   1:  PR[91,3] = PR[90,3] + 124.000;
   1:L PR[91] R[100]mm/sec CNT100;
   1:  PR[91,1] = PR[90,1] + 30.028;
   1:  PR[91,2] = PR[90,2] + -32.892;
   1:  PR[91,3] = PR[90,3] + 124.033;
   1:L PR[91] R[100]mm/sec CNT100;
   1:  PR[91,1] = PR[90,1] + 35.963;
   1:  PR[91,2] = PR[90,2] + -33.565;
   1:  PR[91,3] = PR[90,3] + 124.037;
   1:L PR[91] R[100]mm/sec CNT100;
   1:  PR[91,1] = PR[90,1] + 39.201;
   1:  PR[91,2] = PR[90,2] + -33.483;
   1:  PR[91,3] = PR[90,3] + 124.069;
   1:L PR[91] R[100]mm/sec CNT100;
   1:  PR[91,1] = PR[90,1] + 41.469;
   1:  PR[91,2] = PR[90,2] + -33.515;
   1:  PR[91,3] = PR[90,3] + 124.087;
   1:L PR[91] R[100]mm/sec CNT100;
   1:  PR[91,1] = PR[90,1] + 46.063;
   1:  PR[91,2] = PR[90,2] + -32.960;
   1:  PR[91,3] = PR[90,3] + 124.100;
   1:L PR[91] R[100]mm/sec CNT100;
   1:  PR[91,1] = PR[90,1] + 51.110;
   1:  PR[91,2] = PR[90,2] + -31.758;
   1:  PR[91,3] = PR[90,3] + 124.125;
   1:L PR[91] R[100]mm/sec CNT100;
   1:  PR[91,1] = PR[90,1] + 55.094;
   1:  PR[91,2] = PR[90,2] + -30.275;
   1:  PR[91,3] = PR[90,3] + 124.154;
   1:L PR[91] R[100]mm/sec CNT100;
   1:  PR[91,1] = PR[90,1] + 56.952;
   1:  PR[91,2] = PR[90,2] + -29.564;
   1:  PR[91,3] = PR[90,3] + 124.177;
   1:L PR[91] R[100]mm/sec CNT100;
   1:  PR[91,1] = PR[90,1] + 60.634;
   1:  PR[91,2] = PR[90,2] + -27.680;
   1:  PR[91,3] = PR[90,3] + 124.188;
   1:L PR[91] R[100]mm/sec CNT100;
   1:  PR[91,1] = PR[90,1] + 63.603;
   1:  PR[91,2] = PR[90,2] + -25.642;
   1:  PR[91,3] = PR[90,3] + 124.211;
   1:L PR[91] R[100]mm/sec CNT100;
   1:  PR[91,1] = PR[90,1] + 65.936;
   1:  PR[91,2] = PR[90,2] + -23.984;
   1:  PR[91,3] = PR[90,3] + 124.231;
   1:L PR[91] R[100]mm/sec CNT100;
   1:  PR[91,1] = PR[90,1] + 68.476;
   1:  PR[91,2] = PR[90,2] + -21.706;
   1:  PR[91,3] = PR[90,3] + 124.247;
   1:L PR[91] R[100]mm/sec CNT100;
   1:  PR[91,1] = PR[90,1] + 70.481;
   1:  PR[91,2] = PR[90,2] + -19.318;
   1:  PR[91,3] = PR[90,3] + 124.265;
   1:L PR[91] R[100]mm/sec CNT100;
   1:  PR[91,1] = PR[90,1] + 72.483;
   1:  PR[91,2] = PR[90,2] + -16.900;
   1:  PR[91,3] = PR[90,3] + 124.282;
   1:L PR[91] R[100]mm/sec CNT100;
   1:  PR[91,1] = PR[90,1] + 74.009;
   1:  PR[91,2] = PR[90,2] + -14.439;
   1:  PR[91,3] = PR[90,3] + 124.300;
   1:L PR[91] R[100]mm/sec CNT100;
   1:  PR[91,1] = PR[90,1] + 75.113;
   1:  PR[91,2] = PR[90,2] + -11.830;
   1:  PR[91,3] = PR[90,3] + 124.316;
   1:L PR[91] R[100]mm/sec CNT100;
   1:  PR[91,1] = PR[90,1] + 76.392;
   1:  PR[91,2] = PR[90,2] + -8.966;
   1:  PR[91,3] = PR[90,3] + 124.331;
   1:L PR[91] R[100]mm/sec CNT100;
   1:  PR[91,1] = PR[90,1] + 77.017;
   1:  PR[91,2] = PR[90,2] + -6.453;
   1:  PR[91,3] = PR[90,3] + 124.349;
   1:L PR[91] R[100]mm/sec CNT100;
   1:  PR[91,1] = PR[90,1] + 77.241;
   1:  PR[91,2] = PR[90,2] + -3.694;
   1:  PR[91,3] = PR[90,3] + 124.363;
   1:L PR[91] R[100]mm/sec CNT100;
   1:  PR[91,1] = PR[90,1] + 77.670;
   1:  PR[91,2] = PR[90,2] + -0.670;
   1:  PR[91,3] = PR[90,3] + 124.378;
   1:L PR[91] R[100]mm/sec CNT100;
   1:  PR[91,1] = PR[90,1] + 77.457;
   1:  PR[91,2] = PR[90,2] + 1.932;
   1:  PR[91,3] = PR[90,3] + 124.395;
   1:L PR[91] R[100]mm/sec CNT100;
   1:  PR[91,1] = PR[90,1] + 77.031;
   1:  PR[91,2] = PR[90,2] + 4.936;
   1:  PR[91,3] = PR[90,3] + 124.409;
   1:L PR[91] R[100]mm/sec CNT100;
   1:  PR[91,1] = PR[90,1] + 76.387;
   1:  PR[91,2] = PR[90,2] + 7.526;
   1:  PR[91,3] = PR[90,3] + 124.426;
   1:L PR[91] R[100]mm/sec CNT100;
   1:  PR[91,1] = PR[90,1] + 75.251;
   1:  PR[91,2] = PR[90,2] + 10.206;
   1:  PR[91,3] = PR[90,3] + 124.441;
   1:L PR[91] R[100]mm/sec CNT100;
   1:  PR[91,1] = PR[90,1] + 74.019;
   1:  PR[91,2] = PR[90,2] + 12.964;
   1:  PR[91,3] = PR[90,3] + 124.457;
   1:L PR[91] R[100]mm/sec CNT100;
   1:  PR[91,1] = PR[90,1] + 72.487;
   1:  PR[91,2] = PR[90,2] + 15.435;
   1:  PR[91,3] = PR[90,3] + 124.473;
   1:L PR[91] R[100]mm/sec CNT100;
   1:  PR[91,1] = PR[90,1] + 70.311;
   1:  PR[91,2] = PR[90,2] + 18.030;
   1:  PR[91,3] = PR[90,3] + 124.489;
   1:L PR[91] R[100]mm/sec CNT100;
   1:  PR[91,1] = PR[90,1] + 68.471;
   1:  PR[91,2] = PR[90,2] + 20.251;
   1:  PR[91,3] = PR[90,3] + 124.508;
   1:L PR[91] R[100]mm/sec CNT100;
   1:  PR[91,1] = PR[90,1] + 65.947;
   1:  PR[91,2] = PR[90,2] + 22.515;
   1:  PR[91,3] = PR[90,3] + 124.524;
   1:L PR[91] R[100]mm/sec CNT100;
   1:  PR[91,1] = PR[90,1] + 62.564;
   1:  PR[91,2] = PR[90,2] + 24.848;
   1:  PR[91,3] = PR[90,3] + 124.543;
   1:L PR[91] R[100]mm/sec CNT100;
   1:  PR[91,1] = PR[90,1] + 60.621;
   1:  PR[91,2] = PR[90,2] + 26.228;
   1:  PR[91,3] = PR[90,3] + 124.565;
   1:L PR[91] R[100]mm/sec CNT100;
   1:  PR[91,1] = PR[90,1] + 56.958;
   1:  PR[91,2] = PR[90,2] + 28.102;
   1:  PR[91,3] = PR[90,3] + 124.578;
   1:L PR[91] R[100]mm/sec CNT100;
   1:  PR[91,1] = PR[90,1] + 51.107;
   1:  PR[91,2] = PR[90,2] + 30.300;
   1:  PR[91,3] = PR[90,3] + 124.601;
   1:L PR[91] R[100]mm/sec CNT100;
   1:  PR[91,1] = PR[90,1] + 46.063;
   1:  PR[91,2] = PR[90,2] + 31.501;
   1:  PR[91,3] = PR[90,3] + 124.635;
   1:L PR[91] R[100]mm/sec CNT100;
   1:  PR[91,1] = PR[90,1] + 41.435;
   1:  PR[91,2] = PR[90,2] + 32.060;
   1:  PR[91,3] = PR[90,3] + 124.664;
   1:L PR[91] R[100]mm/sec CNT100;
   1:  PR[91,1] = PR[90,1] + 38.543;
   1:  PR[91,2] = PR[90,2] + 32.110;
   1:  PR[91,3] = PR[90,3] + 124.690;
   1:L PR[91] R[100]mm/sec CNT100;
   1:  PR[91,1] = PR[90,1] + 35.988;
   1:  PR[91,3] = PR[90,3] + 124.705;
   1:L PR[91] R[100]mm/sec CNT100;
   1:  PR[91,1] = PR[90,1] + 30.052;
   1:  PR[91,2] = PR[90,2] + 31.436;
   1:  PR[91,3] = PR[90,3] + 124.720;
   1:L PR[91] R[100]mm/sec CNT100;
   1:  PR[91,1] = PR[90,1] + 26.924;
   1:  PR[91,2] = PR[90,2] + 30.690;
   1:  PR[91,3] = PR[90,3] + 124.752;
   1:L PR[91] R[100]mm/sec CNT100;
   1:  PR[91,1] = PR[90,1] + 23.579;
   1:  PR[91,2] = PR[90,2] + 29.862;
   1:  PR[91,3] = PR[90,3] + 124.770;
   1:L PR[91] R[100]mm/sec CNT100;
   1:  PR[91,1] = PR[90,1] + 21.241;
   1:  PR[91,2] = PR[90,2] + 29.032;
   1:  PR[91,3] = PR[90,3] + 124.789;
   1:L PR[91] R[100]mm/sec CNT100;
   1:  PR[91,1] = PR[90,1] + 17.734;
   1:  PR[91,2] = PR[90,2] + 27.634;
   1:  PR[91,3] = PR[90,3] + 124.803;
   1:L PR[91] R[100]mm/sec CNT100;
   1:  PR[91,1] = PR[90,1] + 13.334;
   1:  PR[91,2] = PR[90,2] + 25.268;
   1:  PR[91,3] = PR[90,3] + 124.824;
   1:L PR[91] R[100]mm/sec CNT100;
   1:  PR[91,1] = PR[90,1] + 11.692;
   1:  PR[91,2] = PR[90,2] + 24.472;
   1:  PR[91,3] = PR[90,3] + 124.851;
   1:L PR[91] R[100]mm/sec CNT100;
   1:  PR[91,1] = PR[90,1] + 5.360;
   1:  PR[91,2] = PR[90,2] + 20.090;
   1:  PR[91,3] = PR[90,3] + 124.861;
   1:L PR[91] R[100]mm/sec CNT100;
   1:  PR[91,1] = PR[90,1] + 2.591;
   1:  PR[91,2] = PR[90,2] + 17.341;
   1:  PR[91,3] = PR[90,3] + 124.904;
   1:L PR[91] R[100]mm/sec CNT100;
   1:  PR[91,1] = PR[90,1] + 0.096;
   1:  PR[91,2] = PR[90,2] + 15.373;
   1:  PR[91,3] = PR[90,3] + 124.925;
   1:L PR[91] R[100]mm/sec CNT100;
   1:  PR[91,1] = PR[90,1] + -1.259;
   1:  PR[91,2] = PR[90,2] + 13.948;
   1:  PR[91,3] = PR[90,3] + 124.942;
   1:L PR[91] R[100]mm/sec CNT100;
   1:  PR[91,1] = PR[90,1] + -3.418;
   1:  PR[91,2] = PR[90,2] + 11.410;
   1:  PR[91,3] = PR[90,3] + 124.953;
   1:L PR[91] R[100]mm/sec CNT100;
   1:  PR[91,1] = PR[90,1] + -5.567;
   1:  PR[91,2] = PR[90,2] + 8.096;
   1:  PR[91,3] = PR[90,3] + 124.972;
   1:L PR[91] R[100]mm/sec CNT100;
   1:  PR[91,1] = PR[90,1] + -5.693;
   1:  PR[91,2] = PR[90,2] + 7.837;
   1:  PR[91,3] = PR[90,3] + 124.993;
   1:L PR[91] R[100]mm/sec CNT100;
   1:  PR[91] = PR[90];
   1:  PR[91,1] = PR[90,1] + -5.574;
   1:  PR[91,2] = PR[90,2] + 3.809;
   1:  PR[91,3] = PR[90,3] + 126.295;
   1:L PR[91] R[100]mm/sec CNT100;
   1:  PR[91,1] = PR[90,1] + -6.141;
   1:  PR[91,2] = PR[90,2] + -0.559;
   1:  PR[91,3] = PR[90,3] + 125.014;
   1:L PR[91] R[100]mm/sec CNT100;
   1:  PR[91,1] = PR[90,1] + -6.172;
   1:  PR[91,2] = PR[90,2] + -0.756;
   1:  PR[91,3] = PR[90,3] + 125.038;
   1:L PR[91] R[100]mm/sec CNT100;
   1:  PR[91,1] = PR[90,1] + -5.675;
   1:  PR[91,2] = PR[90,2] + -4.661;
   1:  PR[91,3] = PR[90,3] + 125.039;
   1:L PR[91] R[100]mm/sec CNT100;
   1:  PR[91,1] = PR[90,1] + -5.583;
   1:  PR[91,2] = PR[90,2] + -5.243;
   1:  PR[91,3] = PR[90,3] + 125.061;
   1:L PR[91] R[100]mm/sec CNT100;
   1:  PR[91,1] = PR[90,1] + -4.357;
   1:  PR[91,2] = PR[90,2] + -8.470;
   1:  PR[91,3] = PR[90,3] + 125.065;
   1:L PR[91] R[100]mm/sec CNT100;
   1:  PR[91,1] = PR[90,1] + -3.471;
   1:  PR[91,2] = PR[90,2] + -10.288;
   1:  PR[91,3] = PR[90,3] + 125.084;
   1:L PR[91] R[100]mm/sec CNT100;
   1:  PR[91,1] = PR[90,1] + -2.114;
   1:  PR[91,2] = PR[90,2] + -12.382;
   1:  PR[91,3] = PR[90,3] + 125.095;
   1:L PR[91] R[100]mm/sec CNT100;
   1:  PR[91,1] = PR[90,1] + 1.492;
   1:  PR[91,2] = PR[90,2] + -16.619;
   1:  PR[91,3] = PR[90,3] + 125.109;
   1:L PR[91] R[100]mm/sec CNT100;
   1:  PR[91,1] = PR[90,1] + 1.499;
   1:  PR[91,2] = PR[90,2] + -16.626;
   1:  PR[91,3] = PR[90,3] + 125.139;
   1:L PR[91] R[100]mm/sec CNT100;
   1:  PR[91,1] = PR[90,1] + 1.719;
   1:  PR[91,2] = PR[90,2] + -16.800;
   1:  PR[91,3] = PR[90,3] + 125.140;
   1:L PR[91] R[100]mm/sec CNT100;
   1:  PR[91,1] = PR[90,1] + 6.651;
   1:  PR[91,2] = PR[90,2] + -21.698;
   1:  PR[91,3] = PR[90,3] + 125.141;
   1:L PR[91] R[100]mm/sec CNT100;
   1:  PR[91,1] = PR[90,1] + 12.464;
   1:  PR[91,2] = PR[90,2] + -25.715;
   1:  PR[91,3] = PR[90,3] + 125.180;
   1:L PR[91] R[100]mm/sec CNT100;
   1:  PR[91,1] = PR[90,1] + 12.954;
   1:  PR[91,2] = PR[90,2] + -26.093;
   1:  PR[91,3] = PR[90,3] + 125.219;
   1:L PR[91] R[100]mm/sec CNT100;
   1:  PR[91,1] = PR[90,1] + 13.257;
   1:  PR[91,2] = PR[90,2] + -26.269;
   1:  PR[91,3] = PR[90,3] + 125.222;
   1:L PR[91] R[100]mm/sec CNT100;
   1:  PR[91,1] = PR[90,1] + 18.422;
   1:  PR[91,2] = PR[90,2] + -29.047;
   1:  PR[91,3] = PR[90,3] + 125.224;
   1:L PR[91] R[100]mm/sec CNT100;
   1:  PR[91,1] = PR[90,1] + 23.423;
   1:  PR[91,2] = PR[90,2] + -31.043;
   1:  PR[91,3] = PR[90,3] + 125.257;
   1:L PR[91] R[100]mm/sec CNT100;
   1:  PR[91,1] = PR[90,1] + 24.234;
   1:  PR[91,2] = PR[90,2] + -31.331;
   1:  PR[91,3] = PR[90,3] + 125.286;
   1:L PR[91] R[100]mm/sec CNT100;
   1:  PR[91,1] = PR[90,1] + 29.647;
   1:  PR[91,2] = PR[90,2] + -32.658;
   1:  PR[91,3] = PR[90,3] + 125.291;
   1:L PR[91] R[100]mm/sec CNT100;
   1:  PR[91,1] = PR[90,1] + 30.937;
   1:  PR[91,2] = PR[90,2] + -32.945;
   1:  PR[91,3] = PR[90,3] + 125.322;
   1:L PR[91] R[100]mm/sec CNT100;
   1:  PR[91,1] = PR[90,1] + 36.646;
   1:  PR[91,2] = PR[90,2] + -33.595;
   1:  PR[91,3] = PR[90,3] + 125.329;
   1:L PR[91] R[100]mm/sec CNT100;
   1:  PR[91,1] = PR[90,1] + 38.964;
   1:  PR[91,2] = PR[90,2] + -33.537;
   1:  PR[91,3] = PR[90,3] + 125.361;
   1:L PR[91] R[100]mm/sec CNT100;
   1:  PR[91,1] = PR[90,1] + 41.893;
   1:  PR[91,2] = PR[90,2] + -33.577;
   1:  PR[91,3] = PR[90,3] + 125.374;
   1:L PR[91] R[100]mm/sec CNT100;
   1:  PR[91,1] = PR[90,1] + 46.843;
   1:  PR[91,2] = PR[90,2] + -32.976;
   1:  PR[91,3] = PR[90,3] + 125.390;
   1:L PR[91] R[100]mm/sec CNT100;
   1:  PR[91,1] = PR[90,1] + 47.163;
   1:  PR[91,2] = PR[90,2] + -32.917;
   1:  PR[91,3] = PR[90,3] + 125.418;
   1:L PR[91] R[100]mm/sec CNT100;
   1:  PR[91,1] = PR[90,1] + 51.875;
   1:  PR[91,2] = PR[90,2] + -31.789;
   1:  PR[91,3] = PR[90,3] + 125.420;
   1:L PR[91] R[100]mm/sec CNT100;
   1:  PR[91,1] = PR[90,1] + 55.644;
   1:  PR[91,2] = PR[90,2] + -30.386;
   1:  PR[91,3] = PR[90,3] + 125.447;
   1:L PR[91] R[100]mm/sec CNT100;
   1:  PR[91,1] = PR[90,1] + 57.968;
   1:  PR[91,2] = PR[90,2] + -29.496;
   1:  PR[91,3] = PR[90,3] + 125.469;
   1:L PR[91] R[100]mm/sec CNT100;
   1:  PR[91,1] = PR[90,1] + 61.445;
   1:  PR[91,2] = PR[90,2] + -27.718;
   1:  PR[91,3] = PR[90,3] + 125.483;
   1:L PR[91] R[100]mm/sec CNT100;
   1:  PR[91,1] = PR[90,1] + 64.251;
   1:  PR[91,2] = PR[90,2] + -25.791;
   1:  PR[91,3] = PR[90,3] + 125.504;
   1:L PR[91] R[100]mm/sec CNT100;
   1:  PR[91,1] = PR[90,1] + 66.907;
   1:  PR[91,2] = PR[90,2] + -23.903;
   1:  PR[91,3] = PR[90,3] + 125.523;
   1:L PR[91] R[100]mm/sec CNT100;
   1:  PR[91,1] = PR[90,1] + 69.303;
   1:  PR[91,2] = PR[90,2] + -21.754;
   1:  PR[91,3] = PR[90,3] + 125.541;
   1:L PR[91] R[100]mm/sec CNT100;
   1:  PR[91,1] = PR[90,1] + 71.198;
   1:  PR[91,2] = PR[90,2] + -19.499;
   1:  PR[91,3] = PR[90,3] + 125.559;
   1:L PR[91] R[100]mm/sec CNT100;
   1:  PR[91,1] = PR[90,1] + 73.408;
   1:  PR[91,2] = PR[90,2] + -16.830;
   1:  PR[91,3] = PR[90,3] + 125.575;
   1:L PR[91] R[100]mm/sec CNT100;
   1:  PR[91,1] = PR[90,1] + 74.844;
   1:  PR[91,2] = PR[90,2] + -14.512;
   1:  PR[91,3] = PR[90,3] + 125.594;
   1:L PR[91] R[100]mm/sec CNT100;
   1:  PR[91,1] = PR[90,1] + 75.888;
   1:  PR[91,2] = PR[90,2] + -12.046;
   1:  PR[91,3] = PR[90,3] + 125.610;
   1:L PR[91] R[100]mm/sec CNT100;
   1:  PR[91,1] = PR[90,1] + 77.282;
   1:  PR[91,2] = PR[90,2] + -8.925;
   1:  PR[91,3] = PR[90,3] + 125.624;
   1:L PR[91] R[100]mm/sec CNT100;
   1:  PR[91,1] = PR[90,1] + 77.869;
   1:  PR[91,2] = PR[90,2] + -6.562;
   1:  PR[91,3] = PR[90,3] + 125.643;
   1:L PR[91] R[100]mm/sec CNT100;
   1:  PR[91,1] = PR[90,1] + 78.081;
   1:  PR[91,2] = PR[90,2] + -3.954;
   1:  PR[91,3] = PR[90,3] + 125.657;
   1:L PR[91] R[100]mm/sec CNT100;
   1:  PR[91,1] = PR[90,1] + 78.547;
   1:  PR[91,2] = PR[90,2] + -0.670;
   1:  PR[91,3] = PR[90,3] + 125.671;
   1:L PR[91] R[100]mm/sec CNT100;
   1:  PR[91,1] = PR[90,1] + 78.347;
   1:  PR[91,2] = PR[90,2] + 1.780;
   1:  PR[91,3] = PR[90,3] + 125.690;
   1:L PR[91] R[100]mm/sec CNT100;
   1:  PR[91,1] = PR[90,1] + 77.883;
   1:  PR[91,2] = PR[90,2] + 5.046;
   1:  PR[91,3] = PR[90,3] + 125.703;
   1:L PR[91] R[100]mm/sec CNT100;
   1:  PR[91,1] = PR[90,1] + 77.277;
   1:  PR[91,2] = PR[90,2] + 7.485;
   1:  PR[91,3] = PR[90,3] + 125.722;
   1:L PR[91] R[100]mm/sec CNT100;
   1:  PR[91,1] = PR[90,1] + 76.204;
   1:  PR[91,2] = PR[90,2] + 10.015;
   1:  PR[91,3] = PR[90,3] + 125.735;
   1:L PR[91] R[100]mm/sec CNT100;
   1:  PR[91,1] = PR[90,1] + 74.854;
   1:  PR[91,2] = PR[90,2] + 13.036;
   1:  PR[91,3] = PR[90,3] + 125.751;
   1:L PR[91] R[100]mm/sec CNT100;
   1:  PR[91,1] = PR[90,1] + 73.411;
   1:  PR[91,2] = PR[90,2] + 15.365;
   1:  PR[91,3] = PR[90,3] + 125.769;
   1:L PR[91] R[100]mm/sec CNT100;
   1:  PR[91,1] = PR[90,1] + 71.354;
   1:  PR[91,2] = PR[90,2] + 17.818;
   1:  PR[91,3] = PR[90,3] + 125.784;
   1:L PR[91] R[100]mm/sec CNT100;
   1:  PR[91,1] = PR[90,1] + 69.298;
   1:  PR[91,2] = PR[90,2] + 20.300;
   1:  PR[91,3] = PR[90,3] + 125.802;
   1:L PR[91] R[100]mm/sec CNT100;
   1:  PR[91,1] = PR[90,1] + 66.918;
   1:  PR[91,2] = PR[90,2] + 22.435;
   1:  PR[91,3] = PR[90,3] + 125.820;
   1:L PR[91] R[100]mm/sec CNT100;
   1:  PR[91,1] = PR[90,1] + 63.719;
   1:  PR[91,2] = PR[90,2] + 24.641;
   1:  PR[91,3] = PR[90,3] + 125.837;
   1:L PR[91] R[100]mm/sec CNT100;
   1:  PR[91,1] = PR[90,1] + 61.431;
   1:  PR[91,2] = PR[90,2] + 26.266;
   1:  PR[91,3] = PR[90,3] + 125.859;
   1:L PR[91] R[100]mm/sec CNT100;
   1:  PR[91,1] = PR[90,1] + 57.975;
   1:  PR[91,2] = PR[90,2] + 28.034;
   1:  PR[91,3] = PR[90,3] + 125.875;
   1:L PR[91] R[100]mm/sec CNT100;
   1:  PR[91,1] = PR[90,1] + 53.451;
   1:  PR[91,2] = PR[90,2] + 29.725;
   1:  PR[91,3] = PR[90,3] + 125.896;
   1:L PR[91] R[100]mm/sec CNT100;
   1:  PR[91,1] = PR[90,1] + 51.866;
   1:  PR[91,2] = PR[90,2] + 30.332;
   1:  PR[91,3] = PR[90,3] + 125.923;
   1:L PR[91] R[100]mm/sec CNT100;
   1:  PR[91,1] = PR[90,1] + 47.163;
   1:  PR[91,2] = PR[90,2] + 31.458;
   1:  PR[91,3] = PR[90,3] + 125.932;
   1:L PR[91] R[100]mm/sec CNT100;
   1:  PR[91,1] = PR[90,1] + 46.843;
   1:  PR[91,2] = PR[90,2] + 31.517;
   1:  PR[91,3] = PR[90,3] + 125.959;
   1:L PR[91] R[100]mm/sec CNT100;
   1:  PR[91,1] = PR[90,1] + 41.861;
   1:  PR[91,2] = PR[90,2] + 32.122;
   1:  PR[91,3] = PR[90,3] + 125.961;
   1:L PR[91] R[100]mm/sec CNT100;
   1:  PR[91,1] = PR[90,1] + 40.847;
   1:  PR[91,2] = PR[90,2] + 32.140;
   1:  PR[91,3] = PR[90,3] + 125.989;
   1:L PR[91] R[100]mm/sec CNT100;
   1:  PR[91,1] = PR[90,1] + 36.672;
   1:  PR[91,3] = PR[90,3] + 125.994;
   1:L PR[91] R[100]mm/sec CNT100;
   1:  PR[91,1] = PR[90,1] + 30.961;
   1:  PR[91,2] = PR[90,2] + 31.489;
   1:  PR[91,3] = PR[90,3] + 126.017;
   1:L PR[91] R[100]mm/sec CNT100;
   1:  PR[91,1] = PR[90,1] + 24.238;
   1:  PR[91,2] = PR[90,2] + 29.873;
   1:  PR[91,3] = PR[90,3] + 126.049;
   1:L PR[91] R[100]mm/sec CNT100;
   1:  PR[91,1] = PR[90,1] + 23.437;
   1:  PR[91,2] = PR[90,2] + 29.589;
   1:  PR[91,3] = PR[90,3] + 126.087;
   1:L PR[91] R[100]mm/sec CNT100;
   1:  PR[91,1] = PR[90,1] + 18.430;
   1:  PR[91,2] = PR[90,2] + 27.592;
   1:  PR[91,3] = PR[90,3] + 126.092;
   1:L PR[91] R[100]mm/sec CNT100;
   1:  PR[91,1] = PR[90,1] + 13.273;
   1:  PR[91,2] = PR[90,2] + 24.819;
   1:  PR[91,3] = PR[90,3] + 126.122;
   1:L PR[91] R[100]mm/sec CNT100;
   1:  PR[91,1] = PR[90,1] + 12.963;
   1:  PR[91,2] = PR[90,2] + 24.639;
   1:  PR[91,3] = PR[90,3] + 126.154;
   1:L PR[91] R[100]mm/sec CNT100;
   1:  PR[91,1] = PR[90,1] + 12.464;
   1:  PR[91,2] = PR[90,2] + 24.255;
   1:  PR[91,3] = PR[90,3] + 126.156;
   1:L PR[91] R[100]mm/sec CNT100;
   1:  PR[91,1] = PR[90,1] + 6.655;
   1:  PR[91,2] = PR[90,2] + 20.242;
   1:  PR[91,3] = PR[90,3] + 126.160;
   1:L PR[91] R[100]mm/sec CNT100;
   1:  PR[91,1] = PR[90,1] + 1.719;
   1:  PR[91,2] = PR[90,2] + 15.341;
   1:  PR[91,3] = PR[90,3] + 126.199;
   1:L PR[91] R[100]mm/sec CNT100;
   1:  PR[91,1] = PR[90,1] + 1.499;
   1:  PR[91,2] = PR[90,2] + 15.168;
   1:  PR[91,3] = PR[90,3] + 126.238;
   1:L PR[91] R[100]mm/sec CNT100;
   1:  PR[91,1] = PR[90,1] + 1.492;
   1:  PR[91,2] = PR[90,2] + 15.160;
   1:  PR[91,3] = PR[90,3] + 126.239;
   1:L PR[91] R[100]mm/sec CNT100;
   1:  PR[91,1] = PR[90,1] + -2.114;
   1:  PR[91,2] = PR[90,2] + 10.923;
   1:L PR[91] R[100]mm/sec CNT100;
   1:  PR[91,1] = PR[90,1] + -3.471;
   1:  PR[91,2] = PR[90,2] + 8.829;
   1:  PR[91,3] = PR[90,3] + 126.270;
   1:L PR[91] R[100]mm/sec CNT100;
   1:  PR[91,1] = PR[90,1] + -4.357;
   1:  PR[91,2] = PR[90,2] + 7.011;
   1:  PR[91,3] = PR[90,3] + 126.284;
   1:L PR[91] R[100]mm/sec CNT100;
   1:  PR[91] = PR[90];
   1:  PR[91,1] = PR[90,1] + -3.791;
   1:  PR[91,2] = PR[90,2] + 4.159;
   1:  PR[91,3] = PR[90,3] + 127.595;
   1:L PR[91] R[100]mm/sec CNT100;
   1:  PR[91,1] = PR[90,1] + -4.159;
   1:  PR[91,2] = PR[90,2] + 1.325;
   1:  PR[91,3] = PR[90,3] + 126.307;
   1:L PR[91] R[100]mm/sec CNT100;
   1:  PR[91,1] = PR[90,1] + -4.481;
   1:  PR[91,2] = PR[90,2] + -0.756;
   1:  PR[91,3] = PR[90,3] + 126.323;
   1:L PR[91] R[100]mm/sec CNT100;
   1:  PR[91,1] = PR[90,1] + -4.146;
   1:  PR[91,2] = PR[90,2] + -3.392;
   1:  PR[91,3] = PR[90,3] + 126.335;
   1:L PR[91] R[100]mm/sec CNT100;
   1:  PR[91,1] = PR[90,1] + -3.801;
   1:  PR[91,2] = PR[90,2] + -5.593;
   1:  PR[91,3] = PR[90,3] + 126.349;
   1:L PR[91] R[100]mm/sec CNT100;
   1:  PR[91,1] = PR[90,1] + -3.021;
   1:  PR[91,2] = PR[90,2] + -7.644;
   1:  PR[91,3] = PR[90,3] + 126.362;
   1:L PR[91] R[100]mm/sec CNT100;
   1:  PR[91,1] = PR[90,1] + -1.375;
   1:  PR[91,2] = PR[90,2] + -11.021;
   1:  PR[91,3] = PR[90,3] + 126.374;
   1:L PR[91] R[100]mm/sec CNT100;
   1:  PR[91,1] = PR[90,1] + -0.809;
   1:  PR[91,2] = PR[90,2] + -11.894;
   1:  PR[91,3] = PR[90,3] + 126.395;
   1:L PR[91] R[100]mm/sec CNT100;
   1:  PR[91,1] = PR[90,1] + 1.116;
   1:  PR[91,2] = PR[90,2] + -14.156;
   1:  PR[91,3] = PR[90,3] + 126.401;
   1:L PR[91] R[100]mm/sec CNT100;
   1:  PR[91,1] = PR[90,1] + 2.964;
   1:  PR[91,2] = PR[90,2] + -16.913;
   1:  PR[91,3] = PR[90,3] + 126.417;
   1:L PR[91] R[100]mm/sec CNT100;
   1:  PR[91,1] = PR[90,1] + 7.943;
   1:  PR[91,2] = PR[90,2] + -21.848;
   1:  PR[91,3] = PR[90,3] + 126.436;
   1:L PR[91] R[100]mm/sec CNT100;
   1:  PR[91,1] = PR[90,1] + 11.325;
   1:  PR[91,2] = PR[90,2] + -24.184;
   1:  PR[91,3] = PR[90,3] + 126.475;
   1:L PR[91] R[100]mm/sec CNT100;
   1:  PR[91,1] = PR[90,1] + 13.694;
   1:  PR[91,2] = PR[90,2] + -26.010;
   1:  PR[91,3] = PR[90,3] + 126.498;
   1:L PR[91] R[100]mm/sec CNT100;
   1:  PR[91,1] = PR[90,1] + 15.507;
   1:  PR[91,2] = PR[90,2] + -27.063;
   1:  PR[91,3] = PR[90,3] + 126.514;
   1:L PR[91] R[100]mm/sec CNT100;
   1:  PR[91,1] = PR[90,1] + 19.120;
   1:  PR[91,2] = PR[90,2] + -29.006;
   1:  PR[91,3] = PR[90,3] + 126.526;
   1:L PR[91] R[100]mm/sec CNT100;
   1:  PR[91,1] = PR[90,1] + 24.945;
   1:  PR[91,2] = PR[90,2] + -31.339;
   1:  PR[91,3] = PR[90,3] + 126.549;
   1:L PR[91] R[100]mm/sec CNT100;
   1:  PR[91,1] = PR[90,1] + 25.097;
   1:  PR[91,2] = PR[90,2] + -31.390;
   1:  PR[91,3] = PR[90,3] + 126.584;
   1:L PR[91] R[100]mm/sec CNT100;
   1:  PR[91,1] = PR[90,1] + 29.956;
   1:  PR[91,2] = PR[90,2] + -32.577;
   1:  PR[91,3] = PR[90,3] + 126.585;
   1:L PR[91] R[100]mm/sec CNT100;
   1:  PR[91,1] = PR[90,1] + 31.846;
   1:  PR[91,2] = PR[90,2] + -32.998;
   1:  PR[91,3] = PR[90,3] + 126.612;
   1:L PR[91] R[100]mm/sec CNT100;
   1:  PR[91,1] = PR[90,1] + 37.329;
   1:  PR[91,2] = PR[90,2] + -33.626;
   1:  PR[91,3] = PR[90,3] + 126.623;
   1:L PR[91] R[100]mm/sec CNT100;
   1:  PR[91,1] = PR[90,1] + 38.727;
   1:  PR[91,2] = PR[90,2] + -33.590;
   1:  PR[91,3] = PR[90,3] + 126.654;
   1:L PR[91] R[100]mm/sec CNT100;
   1:  PR[91,1] = PR[90,1] + 41.492;
   1:  PR[91,2] = PR[90,2] + -33.628;
   1:  PR[91,3] = PR[90,3] + 126.662;
   1:L PR[91] R[100]mm/sec CNT100;
   1:  PR[91,1] = PR[90,1] + 42.530;
   1:  PR[91,2] = PR[90,2] + -33.612;
   1:  PR[91,3] = PR[90,3] + 126.677;
   1:L PR[91] R[100]mm/sec CNT100;
   1:  PR[91,1] = PR[90,1] + 47.573;
   1:  PR[91,2] = PR[90,2] + -32.998;
   1:  PR[91,3] = PR[90,3] + 126.683;
   1:L PR[91] R[100]mm/sec CNT100;
   1:  PR[91,1] = PR[90,1] + 48.201;
   1:  PR[91,2] = PR[90,2] + -32.882;
   1:  PR[91,3] = PR[90,3] + 126.711;
   1:L PR[91] R[100]mm/sec CNT100;
   1:  PR[91,1] = PR[90,1] + 52.642;
   1:  PR[91,2] = PR[90,2] + -31.819;
   1:  PR[91,3] = PR[90,3] + 126.715;
   1:L PR[91] R[100]mm/sec CNT100;
   1:  PR[91,1] = PR[90,1] + 56.194;
   1:  PR[91,2] = PR[90,2] + -30.497;
   1:  PR[91,3] = PR[90,3] + 126.740;
   1:L PR[91] R[100]mm/sec CNT100;
   1:  PR[91,1] = PR[90,1] + 58.984;
   1:  PR[91,2] = PR[90,2] + -29.429;
   1:  PR[91,3] = PR[90,3] + 126.761;
   1:L PR[91] R[100]mm/sec CNT100;
   1:  PR[91,1] = PR[90,1] + 62.255;
   1:  PR[91,2] = PR[90,2] + -27.755;
   1:  PR[91,3] = PR[90,3] + 126.778;
   1:L PR[91] R[100]mm/sec CNT100;
   1:  PR[91,1] = PR[90,1] + 64.899;
   1:  PR[91,2] = PR[90,2] + -25.940;
   1:  PR[91,3] = PR[90,3] + 126.798;
   1:L PR[91] R[100]mm/sec CNT100;
   1:  PR[91,1] = PR[90,1] + 67.879;
   1:  PR[91,2] = PR[90,2] + -23.823;
   1:  PR[91,3] = PR[90,3] + 126.816;
   1:L PR[91] R[100]mm/sec CNT100;
   1:  PR[91,1] = PR[90,1] + 70.131;
   1:  PR[91,2] = PR[90,2] + -21.803;
   1:  PR[91,3] = PR[90,3] + 126.836;
   1:L PR[91] R[100]mm/sec CNT100;
   1:  PR[91,1] = PR[90,1] + 71.915;
   1:  PR[91,2] = PR[90,2] + -19.678;
   1:  PR[91,3] = PR[90,3] + 126.853;
   1:L PR[91] R[100]mm/sec CNT100;
   1:  PR[91,1] = PR[90,1] + 74.332;
   1:  PR[91,2] = PR[90,2] + -16.759;
   1:  PR[91,3] = PR[90,3] + 126.869;
   1:L PR[91] R[100]mm/sec CNT100;
   1:  PR[91,1] = PR[90,1] + 75.680;
   1:  PR[91,2] = PR[90,2] + -14.584;
   1:  PR[91,3] = PR[90,3] + 126.890;
   1:L PR[91] R[100]mm/sec CNT100;
   1:  PR[91,1] = PR[90,1] + 76.662;
   1:  PR[91,2] = PR[90,2] + -12.263;
   1:  PR[91,3] = PR[90,3] + 126.904;
   1:L PR[91] R[100]mm/sec CNT100;
   1:  PR[91,1] = PR[90,1] + 78.171;
   1:  PR[91,2] = PR[90,2] + -8.885;
   1:  PR[91,3] = PR[90,3] + 126.918;
   1:L PR[91] R[100]mm/sec CNT100;
   1:  PR[91,1] = PR[90,1] + 78.721;
   1:  PR[91,2] = PR[90,2] + -6.671;
   1:  PR[91,3] = PR[90,3] + 126.939;
   1:L PR[91] R[100]mm/sec CNT100;
   1:  PR[91,1] = PR[90,1] + 78.921;
   1:  PR[91,2] = PR[90,2] + -4.214;
   1:  PR[91,3] = PR[90,3] + 126.951;
   1:L PR[91] R[100]mm/sec CNT100;
   1:  PR[91,1] = PR[90,1] + 79.424;
   1:  PR[91,2] = PR[90,2] + -0.670;
   1:  PR[91,3] = PR[90,3] + 126.965;
   1:L PR[91] R[100]mm/sec CNT100;
   1:  PR[91,1] = PR[90,1] + 79.236;
   1:  PR[91,2] = PR[90,2] + 1.628;
   1:  PR[91,3] = PR[90,3] + 126.985;
   1:L PR[91] R[100]mm/sec CNT100;
   1:  PR[91,1] = PR[90,1] + 78.736;
   1:  PR[91,2] = PR[90,2] + 5.155;
   1:  PR[91,3] = PR[90,3] + 126.998;
   1:L PR[91] R[100]mm/sec CNT100;
   1:  PR[91,1] = PR[90,1] + 78.166;
   1:  PR[91,2] = PR[90,2] + 7.445;
   1:  PR[91,3] = PR[90,3] + 127.018;
   1:L PR[91] R[100]mm/sec CNT100;
   1:  PR[91,1] = PR[90,1] + 77.157;
   1:  PR[91,2] = PR[90,2] + 9.825;
   1:  PR[91,3] = PR[90,3] + 127.031;
   1:L PR[91] R[100]mm/sec CNT100;
   1:  PR[91,1] = PR[90,1] + 75.690;
   1:  PR[91,2] = PR[90,2] + 13.109;
   1:  PR[91,3] = PR[90,3] + 127.045;
   1:L PR[91] R[100]mm/sec CNT100;
   1:  PR[91,1] = PR[90,1] + 74.335;
   1:  PR[91,2] = PR[90,2] + 15.295;
   1:  PR[91,3] = PR[90,3] + 127.065;
   1:L PR[91] R[100]mm/sec CNT100;
   1:  PR[91,1] = PR[90,1] + 72.398;
   1:  PR[91,2] = PR[90,2] + 17.605;
   1:  PR[91,3] = PR[90,3] + 127.079;
   1:L PR[91] R[100]mm/sec CNT100;
   1:  PR[91,1] = PR[90,1] + 70.125;
   1:  PR[91,2] = PR[90,2] + 20.349;
   1:  PR[91,3] = PR[90,3] + 127.096;
   1:L PR[91] R[100]mm/sec CNT100;
   1:  PR[91,1] = PR[90,1] + 67.889;
   1:  PR[91,2] = PR[90,2] + 22.354;
   1:  PR[91,3] = PR[90,3] + 127.116;
   1:L PR[91] R[100]mm/sec CNT100;
   1:  PR[91,1] = PR[90,1] + 64.873;
   1:  PR[91,2] = PR[90,2] + 24.434;
   1:  PR[91,3] = PR[90,3] + 127.133;
   1:L PR[91] R[100]mm/sec CNT100;
   1:  PR[91,1] = PR[90,1] + 62.241;
   1:  PR[91,2] = PR[90,2] + 26.304;
   1:  PR[91,3] = PR[90,3] + 127.153;
   1:L PR[91] R[100]mm/sec CNT100;
   1:  PR[91,1] = PR[90,1] + 58.991;
   1:  PR[91,2] = PR[90,2] + 27.966;
   1:  PR[91,3] = PR[90,3] + 127.171;
   1:L PR[91] R[100]mm/sec CNT100;
   1:  PR[91,1] = PR[90,1] + 54.724;
   1:  PR[91,2] = PR[90,2] + 29.562;
   1:  PR[91,3] = PR[90,3] + 127.191;
   1:L PR[91] R[100]mm/sec CNT100;
   1:  PR[91,1] = PR[90,1] + 52.632;
   1:  PR[91,2] = PR[90,2] + 30.362;
   1:  PR[91,3] = PR[90,3] + 127.217;
   1:L PR[91] R[100]mm/sec CNT100;
   1:  PR[91,1] = PR[90,1] + 48.201;
   1:  PR[91,2] = PR[90,2] + 31.423;
   1:  PR[91,3] = PR[90,3] + 127.229;
   1:L PR[91] R[100]mm/sec CNT100;
   1:  PR[91,1] = PR[90,1] + 47.574;
   1:  PR[91,2] = PR[90,2] + 31.539;
   1:  PR[91,3] = PR[90,3] + 127.254;
   1:L PR[91] R[100]mm/sec CNT100;
   1:  PR[91,1] = PR[90,1] + 42.405;
   1:  PR[91,2] = PR[90,2] + 32.161;
   1:  PR[91,3] = PR[90,3] + 127.258;
   1:L PR[91] R[100]mm/sec CNT100;
   1:  PR[91,1] = PR[90,1] + 37.353;
   1:  PR[91,2] = PR[90,2] + 32.170;
   1:  PR[91,3] = PR[90,3] + 127.287;
   1:L PR[91] R[100]mm/sec CNT100;
   1:  PR[91,1] = PR[90,1] + 31.866;
   1:  PR[91,2] = PR[90,2] + 31.542;
   1:  PR[91,3] = PR[90,3] + 127.315;
   1:L PR[91] R[100]mm/sec CNT100;
   1:  PR[91,1] = PR[90,1] + 25.101;
   1:  PR[91,2] = PR[90,2] + 29.932;
   1:  PR[91,3] = PR[90,3] + 127.346;
   1:L PR[91] R[100]mm/sec CNT100;
   1:  PR[91,1] = PR[90,1] + 24.952;
   1:  PR[91,2] = PR[90,2] + 29.883;
   1:  PR[91,3] = PR[90,3] + 127.384;
   1:L PR[91] R[100]mm/sec CNT100;
   1:  PR[91,1] = PR[90,1] + 19.128;
   1:  PR[91,2] = PR[90,2] + 27.551;
   1:  PR[91,3] = PR[90,3] + 127.385;
   1:L PR[91] R[100]mm/sec CNT100;
   1:  PR[91,1] = PR[90,1] + 15.521;
   1:  PR[91,2] = PR[90,2] + 25.612;
   1:  PR[91,3] = PR[90,3] + 127.420;
   1:L PR[91] R[100]mm/sec CNT100;
   1:  PR[91,1] = PR[90,1] + 13.701;
   1:  PR[91,2] = PR[90,2] + 24.557;
   1:  PR[91,3] = PR[90,3] + 127.443;
   1:L PR[91] R[100]mm/sec CNT100;
   1:  PR[91,1] = PR[90,1] + 11.324;
   1:  PR[91,2] = PR[90,2] + 22.725;
   1:  PR[91,3] = PR[90,3] + 127.455;
   1:L PR[91] R[100]mm/sec CNT100;
   1:  PR[91,1] = PR[90,1] + 7.949;
   1:  PR[91,2] = PR[90,2] + 20.393;
   1:  PR[91,3] = PR[90,3] + 127.471;
   1:L PR[91] R[100]mm/sec CNT100;
   1:  PR[91,1] = PR[90,1] + 2.965;
   1:  PR[91,2] = PR[90,2] + 15.455;
   1:  PR[91,3] = PR[90,3] + 127.494;
   1:L PR[91] R[100]mm/sec CNT100;
   1:  PR[91,1] = PR[90,1] + 1.116;
   1:  PR[91,2] = PR[90,2] + 12.697;
   1:  PR[91,3] = PR[90,3] + 127.533;
   1:L PR[91] R[100]mm/sec CNT100;
   1:  PR[91,1] = PR[90,1] + -0.809;
   1:  PR[91,2] = PR[90,2] + 10.435;
   1:  PR[91,3] = PR[90,3] + 127.552;
   1:L PR[91] R[100]mm/sec CNT100;
   1:  PR[91,1] = PR[90,1] + -1.375;
   1:  PR[91,2] = PR[90,2] + 9.562;
   1:  PR[91,3] = PR[90,3] + 127.568;
   1:L PR[91] R[100]mm/sec CNT100;
   1:  PR[91,1] = PR[90,1] + -3.021;
   1:  PR[91,2] = PR[90,2] + 6.185;
   1:  PR[91,3] = PR[90,3] + 127.574;
   1:L PR[91] R[100]mm/sec CNT100;
   1:  PR[91] = PR[90];
   1:  PR[91,1] = PR[90,1] + -2.008;
   1:  PR[91,2] = PR[90,2] + 4.509;
   1:  PR[91,3] = PR[90,3] + 128.895;
   1:L PR[91] R[100]mm/sec CNT100;
   1:  PR[91,1] = PR[90,1] + -2.177;
   1:  PR[91,2] = PR[90,2] + 3.210;
   1:  PR[91,3] = PR[90,3] + 127.600;
   1:L PR[91] R[100]mm/sec CNT100;
   1:  PR[91,1] = PR[90,1] + -2.790;
   1:  PR[91,2] = PR[90,2] + -0.756;
   1:  PR[91,3] = PR[90,3] + 127.607;
   1:L PR[91] R[100]mm/sec CNT100;
   1:  PR[91,1] = PR[90,1] + -2.616;
   1:  PR[91,2] = PR[90,2] + -2.123;
   1:  PR[91,3] = PR[90,3] + 127.630;
   1:L PR[91] R[100]mm/sec CNT100;
   1:  PR[91,1] = PR[90,1] + -2.018;
   1:  PR[91,2] = PR[90,2] + -5.942;
   1:  PR[91,3] = PR[90,3] + 127.638;
   1:L PR[91] R[100]mm/sec CNT100;
   1:  PR[91,1] = PR[90,1] + -1.685;
   1:  PR[91,2] = PR[90,2] + -6.818;
   1:  PR[91,3] = PR[90,3] + 127.659;
   1:L PR[91] R[100]mm/sec CNT100;
   1:  PR[91,1] = PR[90,1] + 0.482;
   1:  PR[91,2] = PR[90,2] + -11.264;
   1:  PR[91,3] = PR[90,3] + 127.664;
   1:L PR[91] R[100]mm/sec CNT100;
   1:  PR[91,1] = PR[90,1] + 0.665;
   1:  PR[91,2] = PR[90,2] + -11.740;
   1:  PR[91,3] = PR[90,3] + 127.692;
   1:L PR[91] R[100]mm/sec CNT100;
   1:  PR[91,1] = PR[90,1] + 4.212;
   1:  PR[91,2] = PR[90,2] + -17.031;
   1:  PR[91,3] = PR[90,3] + 127.695;
   1:L PR[91] R[100]mm/sec CNT100;
   1:  PR[91,1] = PR[90,1] + 9.236;
   1:  PR[91,2] = PR[90,2] + -21.997;
   1:  PR[91,3] = PR[90,3] + 127.730;
   1:L PR[91] R[100]mm/sec CNT100;
   1:  PR[91,1] = PR[90,1] + 10.185;
   1:  PR[91,2] = PR[90,2] + -22.654;
   1:  PR[91,3] = PR[90,3] + 127.770;
   1:L PR[91] R[100]mm/sec CNT100;
   1:  PR[91,1] = PR[90,1] + 14.433;
   1:  PR[91,2] = PR[90,2] + -25.928;
   1:  PR[91,3] = PR[90,3] + 127.776;
   1:L PR[91] R[100]mm/sec CNT100;
   1:  PR[91,1] = PR[90,1] + 17.758;
   1:  PR[91,2] = PR[90,2] + -27.857;
   1:  PR[91,3] = PR[90,3] + 127.806;
   1:L PR[91] R[100]mm/sec CNT100;
   1:  PR[91,1] = PR[90,1] + 19.816;
   1:  PR[91,2] = PR[90,2] + -28.964;
   1:  PR[91,3] = PR[90,3] + 127.828;
   1:L PR[91] R[100]mm/sec CNT100;
   1:  PR[91,1] = PR[90,1] + 22.777;
   1:  PR[91,2] = PR[90,2] + -30.146;
   1:  PR[91,3] = PR[90,3] + 127.841;
   1:L PR[91] R[100]mm/sec CNT100;
   1:  PR[91,1] = PR[90,1] + 25.444;
   1:  PR[91,2] = PR[90,2] + -31.241;
   1:  PR[91,3] = PR[90,3] + 127.859;
   1:L PR[91] R[100]mm/sec CNT100;
   1:  PR[91,1] = PR[90,1] + 26.331;
   1:  PR[91,2] = PR[90,2] + -31.535;
   1:  PR[91,3] = PR[90,3] + 127.875;
   1:L PR[91] R[100]mm/sec CNT100;
   1:  PR[91,1] = PR[90,1] + 30.265;
   1:  PR[91,2] = PR[90,2] + -32.496;
   1:  PR[91,3] = PR[90,3] + 127.880;
   1:L PR[91] R[100]mm/sec CNT100;
   1:  PR[91,1] = PR[90,1] + 32.755;
   1:  PR[91,2] = PR[90,2] + -33.051;
   1:  PR[91,3] = PR[90,3] + 127.903;
   1:L PR[91] R[100]mm/sec CNT100;
   1:  PR[91,1] = PR[90,1] + 38.013;
   1:  PR[91,2] = PR[90,2] + -33.656;
   1:  PR[91,3] = PR[90,3] + 127.917;
   1:L PR[91] R[100]mm/sec CNT100;
   1:  PR[91,1] = PR[90,1] + 38.490;
   1:  PR[91,2] = PR[90,2] + -33.644;
   1:  PR[91,3] = PR[90,3] + 127.946;
   1:L PR[91] R[100]mm/sec CNT100;
   1:  PR[91,1] = PR[90,1] + 39.571;
   1:  PR[91,2] = PR[90,2] + -33.659;
   1:  PR[91,3] = PR[90,3] + 127.949;
   1:L PR[91] R[100]mm/sec CNT100;
   1:  PR[91,1] = PR[90,1] + 43.138;
   1:  PR[91,2] = PR[90,2] + -33.626;
   1:  PR[91,3] = PR[90,3] + 127.955;
   1:L PR[91] R[100]mm/sec CNT100;
   1:  PR[91,1] = PR[90,1] + 43.522;
   1:  PR[91,2] = PR[90,2] + -33.603;
   1:  PR[91,3] = PR[90,3] + 127.975;
   1:L PR[91] R[100]mm/sec CNT100;
   1:  PR[91,1] = PR[90,1] + 48.303;
   1:  PR[91,2] = PR[90,2] + -33.020;
   1:  PR[91,3] = PR[90,3] + 127.977;
   1:L PR[91] R[100]mm/sec CNT100;
   1:  PR[91,1] = PR[90,1] + 49.240;
   1:  PR[91,2] = PR[90,2] + -32.847;
   1:  PR[91,3] = PR[90,3] + 128.004;
   1:L PR[91] R[100]mm/sec CNT100;
   1:  PR[91,1] = PR[90,1] + 53.408;
   1:  PR[91,2] = PR[90,2] + -31.849;
   1:  PR[91,3] = PR[90,3] + 128.010;
   1:L PR[91] R[100]mm/sec CNT100;
   1:  PR[91,1] = PR[90,1] + 56.744;
   1:  PR[91,2] = PR[90,2] + -30.608;
   1:  PR[91,3] = PR[90,3] + 128.033;
   1:L PR[91] R[100]mm/sec CNT100;
   1:  PR[91,1] = PR[90,1] + 59.999;
   1:  PR[91,2] = PR[90,2] + -29.361;
   1:  PR[91,3] = PR[90,3] + 128.053;
   1:L PR[91] R[100]mm/sec CNT100;
   1:  PR[91,1] = PR[90,1] + 63.066;
   1:  PR[91,2] = PR[90,2] + -27.793;
   1:  PR[91,3] = PR[90,3] + 128.073;
   1:L PR[91] R[100]mm/sec CNT100;
   1:  PR[91,1] = PR[90,1] + 65.547;
   1:  PR[91,2] = PR[90,2] + -26.089;
   1:  PR[91,3] = PR[90,3] + 128.092;
   1:L PR[91] R[100]mm/sec CNT100;
   1:  PR[91,1] = PR[90,1] + 68.850;
   1:  PR[91,2] = PR[90,2] + -23.742;
   1:  PR[91,3] = PR[90,3] + 128.109;
   1:L PR[91] R[100]mm/sec CNT100;
   1:  PR[91,1] = PR[90,1] + 70.958;
   1:  PR[91,2] = PR[90,2] + -21.851;
   1:  PR[91,3] = PR[90,3] + 128.132;
   1:L PR[91] R[100]mm/sec CNT100;
   1:  PR[91,1] = PR[90,1] + 72.631;
   1:  PR[91,2] = PR[90,2] + -19.859;
   1:  PR[91,3] = PR[90,3] + 128.147;
   1:L PR[91] R[100]mm/sec CNT100;
   1:  PR[91,1] = PR[90,1] + 75.256;
   1:  PR[91,2] = PR[90,2] + -16.689;
   1:  PR[91,3] = PR[90,3] + 128.162;
   1:L PR[91] R[100]mm/sec CNT100;
   1:  PR[91,1] = PR[90,1] + 76.516;
   1:  PR[91,2] = PR[90,2] + -14.657;
   1:  PR[91,3] = PR[90,3] + 128.185;
   1:L PR[91] R[100]mm/sec CNT100;
   1:  PR[91,1] = PR[90,1] + 77.437;
   1:  PR[91,2] = PR[90,2] + -12.479;
   1:  PR[91,3] = PR[90,3] + 128.198;
   1:L PR[91] R[100]mm/sec CNT100;
   1:  PR[91,1] = PR[90,1] + 79.061;
   1:  PR[91,2] = PR[90,2] + -8.844;
   1:  PR[91,3] = PR[90,3] + 128.211;
   1:L PR[91] R[100]mm/sec CNT100;
   1:  PR[91,1] = PR[90,1] + 79.574;
   1:  PR[91,2] = PR[90,2] + -6.781;
   1:  PR[91,3] = PR[90,3] + 128.234;
   1:L PR[91] R[100]mm/sec CNT100;
   1:  PR[91,1] = PR[90,1] + 79.761;
   1:  PR[91,2] = PR[90,2] + -4.475;
   1:  PR[91,3] = PR[90,3] + 128.246;
   1:L PR[91] R[100]mm/sec CNT100;
   1:  PR[91,1] = PR[90,1] + 80.301;
   1:  PR[91,2] = PR[90,2] + -0.670;
   1:  PR[91,3] = PR[90,3] + 128.259;
   1:L PR[91] R[100]mm/sec CNT100;
   1:  PR[91,1] = PR[90,1] + 80.125;
   1:  PR[91,2] = PR[90,2] + 1.476;
   1:  PR[91,3] = PR[90,3] + 128.280;
   1:L PR[91] R[100]mm/sec CNT100;
   1:  PR[91,1] = PR[90,1] + 79.588;
   1:  PR[91,2] = PR[90,2] + 5.264;
   1:  PR[91,3] = PR[90,3] + 128.292;
   1:L PR[91] R[100]mm/sec CNT100;
   1:  PR[91,1] = PR[90,1] + 79.056;
   1:  PR[91,2] = PR[90,2] + 7.404;
   1:  PR[91,3] = PR[90,3] + 128.313;
   1:L PR[91] R[100]mm/sec CNT100;
   1:  PR[91,1] = PR[90,1] + 78.110;
   1:  PR[91,2] = PR[90,2] + 9.635;
   1:  PR[91,3] = PR[90,3] + 128.326;
   1:L PR[91] R[100]mm/sec CNT100;
   1:  PR[91,1] = PR[90,1] + 76.526;
   1:  PR[91,2] = PR[90,2] + 13.181;
   1:  PR[91,3] = PR[90,3] + 128.339;
   1:L PR[91] R[100]mm/sec CNT100;
   1:  PR[91,1] = PR[90,1] + 75.259;
   1:  PR[91,2] = PR[90,2] + 15.225;
   1:  PR[91,3] = PR[90,3] + 128.361;
   1:L PR[91] R[100]mm/sec CNT100;
   1:  PR[91,1] = PR[90,1] + 73.441;
   1:  PR[91,2] = PR[90,2] + 17.392;
   1:  PR[91,3] = PR[90,3] + 128.374;
   1:L PR[91] R[100]mm/sec CNT100;
   1:  PR[91,1] = PR[90,1] + 70.953;
   1:  PR[91,2] = PR[90,2] + 20.397;
   1:  PR[91,3] = PR[90,3] + 128.390;
   1:L PR[91] R[100]mm/sec CNT100;
   1:  PR[91,1] = PR[90,1] + 68.860;
   1:  PR[91,2] = PR[90,2] + 22.274;
   1:  PR[91,3] = PR[90,3] + 128.412;
   1:L PR[91] R[100]mm/sec CNT100;
   1:  PR[91,1] = PR[90,1] + 66.027;
   1:  PR[91,2] = PR[90,2] + 24.227;
   1:  PR[91,3] = PR[90,3] + 128.428;
   1:L PR[91] R[100]mm/sec CNT100;
   1:  PR[91,1] = PR[90,1] + 63.051;
   1:  PR[91,2] = PR[90,2] + 26.341;
   1:  PR[91,3] = PR[90,3] + 128.447;
   1:L PR[91] R[100]mm/sec CNT100;
   1:  PR[91,1] = PR[90,1] + 60.006;
   1:  PR[91,2] = PR[90,2] + 27.899;
   1:  PR[91,3] = PR[90,3] + 128.467;
   1:L PR[91] R[100]mm/sec CNT100;
   1:  PR[91,1] = PR[90,1] + 55.997;
   1:  PR[91,2] = PR[90,2] + 29.398;
   1:  PR[91,3] = PR[90,3] + 128.486;
   1:L PR[91] R[100]mm/sec CNT100;
   1:  PR[91,1] = PR[90,1] + 53.398;
   1:  PR[91,2] = PR[90,2] + 30.393;
   1:  PR[91,3] = PR[90,3] + 128.510;
   1:L PR[91] R[100]mm/sec CNT100;
   1:  PR[91,1] = PR[90,1] + 49.239;
   1:  PR[91,2] = PR[90,2] + 31.389;
   1:  PR[91,3] = PR[90,3] + 128.526;
   1:L PR[91] R[100]mm/sec CNT100;
   1:  PR[91,1] = PR[90,1] + 48.302;
   1:  PR[91,2] = PR[90,2] + 31.562;
   1:  PR[91,3] = PR[90,3] + 128.550;
   1:L PR[91] R[100]mm/sec CNT100;
   1:  PR[91,1] = PR[90,1] + 43.521;
   1:  PR[91,2] = PR[90,2] + 32.144;
   1:  PR[91,3] = PR[90,3] + 128.555;
   1:L PR[91] R[100]mm/sec CNT100;
   1:  PR[91,1] = PR[90,1] + 43.138;
   1:  PR[91,2] = PR[90,2] + 32.167;
   1:  PR[91,3] = PR[90,3] + 128.582;
   1:L PR[91] R[100]mm/sec CNT100;
   1:  PR[91,1] = PR[90,1] + 39.557;
   1:  PR[91,2] = PR[90,2] + 32.200;
   1:  PR[91,3] = PR[90,3] + 128.584;
   1:L PR[91] R[100]mm/sec CNT100;
   1:  PR[91,1] = PR[90,1] + 38.038;
   1:  PR[91,3] = PR[90,3] + 128.604;
   1:L PR[91] R[100]mm/sec CNT100;
   1:  PR[91,1] = PR[90,1] + 32.774;
   1:  PR[91,2] = PR[90,2] + 31.594;
   1:  PR[91,3] = PR[90,3] + 128.613;
   1:L PR[91] R[100]mm/sec CNT100;
   1:  PR[91,1] = PR[90,1] + 28.310;
   1:  PR[91,2] = PR[90,2] + 30.528;
   1:  PR[91,3] = PR[90,3] + 128.642;
   1:L PR[91] R[100]mm/sec CNT100;
   1:  PR[91,1] = PR[90,1] + 26.325;
   1:  PR[91,2] = PR[90,2] + 30.074;
   1:  PR[91,3] = PR[90,3] + 128.668;
   1:L PR[91] R[100]mm/sec CNT100;
   1:  PR[91,1] = PR[90,1] + 25.449;
   1:  PR[91,2] = PR[90,2] + 29.784;
   1:  PR[91,3] = PR[90,3] + 128.679;
   1:L PR[91] R[100]mm/sec CNT100;
   1:  PR[91,1] = PR[90,1] + 22.777;
   1:  PR[91,2] = PR[90,2] + 28.687;
   1:  PR[91,3] = PR[90,3] + 128.685;
   1:L PR[91] R[100]mm/sec CNT100;
   1:  PR[91,1] = PR[90,1] + 19.823;
   1:  PR[91,2] = PR[90,2] + 27.509;
   1:  PR[91,3] = PR[90,3] + 128.701;
   1:L PR[91] R[100]mm/sec CNT100;
   1:  PR[91,1] = PR[90,1] + 17.771;
   1:  PR[91,2] = PR[90,2] + 26.405;
   1:  PR[91,3] = PR[90,3] + 128.718;
   1:L PR[91] R[100]mm/sec CNT100;
   1:  PR[91,1] = PR[90,1] + 14.440;
   1:  PR[91,2] = PR[90,2] + 24.474;
   1:  PR[91,3] = PR[90,3] + 128.731;
   1:L PR[91] R[100]mm/sec CNT100;
   1:  PR[91,1] = PR[90,1] + 10.185;
   1:  PR[91,2] = PR[90,2] + 21.195;
   1:  PR[91,3] = PR[90,3] + 128.753;
   1:L PR[91] R[100]mm/sec CNT100;
   1:  PR[91,1] = PR[90,1] + 9.243;
   1:  PR[91,2] = PR[90,2] + 20.544;
   1:  PR[91,3] = PR[90,3] + 128.783;
   1:L PR[91] R[100]mm/sec CNT100;
   1:  PR[91,1] = PR[90,1] + 4.214;
   1:  PR[91,2] = PR[90,2] + 15.574;
   1:  PR[91,3] = PR[90,3] + 128.789;
   1:L PR[91] R[100]mm/sec CNT100;
   1:  PR[91,1] = PR[90,1] + 0.665;
   1:  PR[91,2] = PR[90,2] + 10.282;
   1:  PR[91,3] = PR[90,3] + 128.829;
   1:L PR[91] R[100]mm/sec CNT100;
   1:  PR[91,1] = PR[90,1] + 0.482;
   1:  PR[91,2] = PR[90,2] + 9.806;
   1:  PR[91,3] = PR[90,3] + 128.865;
   1:L PR[91] R[100]mm/sec CNT100;
   1:  PR[91,1] = PR[90,1] + -1.685;
   1:  PR[91,2] = PR[90,2] + 5.359;
   1:  PR[91,3] = PR[90,3] + 128.867;
   1:L PR[91] R[100]mm/sec CNT100;
   1:  PR[91] = PR[90];
   1:  PR[91,1] = PR[90,1] + -1.100;
   1:  PR[91,2] = PR[90,2] + -0.755;
   1:  PR[91,3] = PR[90,3] + 130.195;
   1:L PR[91] R[100]mm/sec CNT100;
   1:  PR[91,1] = PR[90,1] + -1.087;
   1:  PR[91,2] = PR[90,2] + -0.854;
   1:  PR[91,3] = PR[90,3] + 128.927;
   1:L PR[91] R[100]mm/sec CNT100;
   1:  PR[91,1] = PR[90,1] + -0.251;
   1:  PR[91,2] = PR[90,2] + -6.189;
   1:L PR[91] R[100]mm/sec CNT100;
   1:  PR[91,1] = PR[90,1] + -0.234;
   1:  PR[91,2] = PR[90,2] + -6.315;
   1:  PR[91,3] = PR[90,3] + 128.958;
   1:L PR[91] R[100]mm/sec CNT100;
   1:  PR[91,1] = PR[90,1] + 1.879;
   1:  PR[91,2] = PR[90,2] + -11.822;
   1:L PR[91] R[100]mm/sec CNT100;
   1:  PR[91,1] = PR[90,1] + 5.460;
   1:  PR[91,2] = PR[90,2] + -17.149;
   1:  PR[91,3] = PR[90,3] + 128.991;
   1:L PR[91] R[100]mm/sec CNT100;
   1:  PR[91,1] = PR[90,1] + 9.311;
   1:  PR[91,2] = PR[90,2] + -20.952;
   1:  PR[91,3] = PR[90,3] + 129.027;
   1:L PR[91] R[100]mm/sec CNT100;
   1:  PR[91,1] = PR[90,1] + 10.345;
   1:  PR[91,2] = PR[90,2] + -22.094;
   1:  PR[91,3] = PR[90,3] + 129.058;
   1:L PR[91] R[100]mm/sec CNT100;
   1:  PR[91,1] = PR[90,1] + 11.008;
   1:  PR[91,2] = PR[90,2] + -22.635;
   1:  PR[91,3] = PR[90,3] + 129.066;
   1:L PR[91] R[100]mm/sec CNT100;
   1:  PR[91,1] = PR[90,1] + 15.173;
   1:  PR[91,2] = PR[90,2] + -25.846;
   1:  PR[91,3] = PR[90,3] + 129.071;
   1:L PR[91] R[100]mm/sec CNT100;
   1:  PR[91,1] = PR[90,1] + 20.008;
   1:  PR[91,2] = PR[90,2] + -28.651;
   1:  PR[91,3] = PR[90,3] + 129.101;
   1:L PR[91] R[100]mm/sec CNT100;
   1:  PR[91,1] = PR[90,1] + 20.520;
   1:  PR[91,2] = PR[90,2] + -28.927;
   1:  PR[91,3] = PR[90,3] + 129.132;
   1:L PR[91] R[100]mm/sec CNT100;
   1:  PR[91,1] = PR[90,1] + 25.932;
   1:  PR[91,2] = PR[90,2] + -31.139;
   1:  PR[91,3] = PR[90,3] + 129.135;
   1:L PR[91] R[100]mm/sec CNT100;
   1:  PR[91,1] = PR[90,1] + 27.565;
   1:  PR[91,2] = PR[90,2] + -31.680;
   1:  PR[91,3] = PR[90,3] + 129.168;
   1:L PR[91] R[100]mm/sec CNT100;
   1:  PR[91,1] = PR[90,1] + 30.574;
   1:  PR[91,2] = PR[90,2] + -32.416;
   1:  PR[91,3] = PR[90,3] + 129.178;
   1:L PR[91] R[100]mm/sec CNT100;
   1:  PR[91,1] = PR[90,1] + 33.664;
   1:  PR[91,2] = PR[90,2] + -33.104;
   1:  PR[91,3] = PR[90,3] + 129.195;
   1:L PR[91] R[100]mm/sec CNT100;
   1:  PR[91,1] = PR[90,1] + 37.847;
   1:  PR[91,2] = PR[90,2] + -33.587;
   1:  PR[91,3] = PR[90,3] + 129.213;
   1:L PR[91] R[100]mm/sec CNT100;
   1:  PR[91,1] = PR[90,1] + 38.818;
   1:  PR[91,2] = PR[90,2] + -33.678;
   1:  PR[91,3] = PR[90,3] + 129.236;
   1:L PR[91] R[100]mm/sec CNT100;
   1:  PR[91,1] = PR[90,1] + 43.820;
   1:  PR[91,2] = PR[90,2] + -33.633;
   1:  PR[91,3] = PR[90,3] + 129.242;
   1:L PR[91] R[100]mm/sec CNT100;
   1:  PR[91,1] = PR[90,1] + 44.559;
   1:  PR[91,2] = PR[90,2] + -33.588;
   1:  PR[91,3] = PR[90,3] + 129.270;
   1:L PR[91] R[100]mm/sec CNT100;
   1:  PR[91,1] = PR[90,1] + 49.033;
   1:  PR[91,2] = PR[90,2] + -33.042;
   1:  PR[91,3] = PR[90,3] + 129.274;
   1:L PR[91] R[100]mm/sec CNT100;
   1:  PR[91,1] = PR[90,1] + 50.278;
   1:  PR[91,2] = PR[90,2] + -32.813;
   1:  PR[91,3] = PR[90,3] + 129.299;
   1:L PR[91] R[100]mm/sec CNT100;
   1:  PR[91,1] = PR[90,1] + 54.175;
   1:  PR[91,2] = PR[90,2] + -31.880;
   1:  PR[91,3] = PR[90,3] + 129.306;
   1:L PR[91] R[100]mm/sec CNT100;
   1:  PR[91,1] = PR[90,1] + 57.294;
   1:  PR[91,2] = PR[90,2] + -30.718;
   1:  PR[91,3] = PR[90,3] + 129.329;
   1:L PR[91] R[100]mm/sec CNT100;
   1:  PR[91,1] = PR[90,1] + 61.015;
   1:  PR[91,2] = PR[90,2] + -29.294;
   1:  PR[91,3] = PR[90,3] + 129.348;
   1:L PR[91] R[100]mm/sec CNT100;
   1:  PR[91,1] = PR[90,1] + 63.876;
   1:  PR[91,2] = PR[90,2] + -27.830;
   1:  PR[91,3] = PR[90,3] + 129.370;
   1:L PR[91] R[100]mm/sec CNT100;
   1:  PR[91,1] = PR[90,1] + 66.195;
   1:  PR[91,2] = PR[90,2] + -26.238;
   1:  PR[91,3] = PR[90,3] + 129.388;
   1:L PR[91] R[100]mm/sec CNT100;
   1:  PR[91,1] = PR[90,1] + 69.821;
   1:  PR[91,2] = PR[90,2] + -23.661;
   1:  PR[91,3] = PR[90,3] + 129.404;
   1:L PR[91] R[100]mm/sec CNT100;
   1:  PR[91,1] = PR[90,1] + 71.785;
   1:  PR[91,2] = PR[90,2] + -21.900;
   1:  PR[91,3] = PR[90,3] + 129.429;
   1:L PR[91] R[100]mm/sec CNT100;
   1:  PR[91,1] = PR[90,1] + 73.347;
   1:  PR[91,2] = PR[90,2] + -20.040;
   1:  PR[91,3] = PR[90,3] + 129.443;
   1:L PR[91] R[100]mm/sec CNT100;
   1:  PR[91,1] = PR[90,1] + 76.180;
   1:  PR[91,2] = PR[90,2] + -16.618;
   1:  PR[91,3] = PR[90,3] + 129.457;
   1:L PR[91] R[100]mm/sec CNT100;
   1:  PR[91,1] = PR[90,1] + 77.351;
   1:  PR[91,2] = PR[90,2] + -14.729;
   1:  PR[91,3] = PR[90,3] + 129.482;
   1:L PR[91] R[100]mm/sec CNT100;
   1:  PR[91,1] = PR[90,1] + 78.212;
   1:  PR[91,2] = PR[90,2] + -12.696;
   1:  PR[91,3] = PR[90,3] + 129.494;
   1:L PR[91] R[100]mm/sec CNT100;
   1:  PR[91,1] = PR[90,1] + 79.950;
   1:  PR[91,2] = PR[90,2] + -8.803;
   1:  PR[91,3] = PR[90,3] + 129.507;
   1:L PR[91] R[100]mm/sec CNT100;
   1:  PR[91,1] = PR[90,1] + 80.426;
   1:  PR[91,2] = PR[90,2] + -6.890;
   1:  PR[91,3] = PR[90,3] + 129.531;
   1:L PR[91] R[100]mm/sec CNT100;
   1:  PR[91,1] = PR[90,1] + 80.601;
   1:  PR[91,2] = PR[90,2] + -4.735;
   1:  PR[91,3] = PR[90,3] + 129.542;
   1:L PR[91] R[100]mm/sec CNT100;
   1:  PR[91,1] = PR[90,1] + 81.178;
   1:  PR[91,2] = PR[90,2] + -0.670;
   1:  PR[91,3] = PR[90,3] + 129.554;
   1:L PR[91] R[100]mm/sec CNT100;
   1:  PR[91,1] = PR[90,1] + 81.015;
   1:  PR[91,2] = PR[90,2] + 1.324;
   1:  PR[91,3] = PR[90,3] + 129.577;
   1:L PR[91] R[100]mm/sec CNT100;
   1:  PR[91,1] = PR[90,1] + 80.440;
   1:  PR[91,2] = PR[90,2] + 5.374;
   1:  PR[91,3] = PR[90,3] + 129.588;
   1:L PR[91] R[100]mm/sec CNT100;
   1:  PR[91,1] = PR[90,1] + 79.945;
   1:  PR[91,2] = PR[90,2] + 7.364;
   1:  PR[91,3] = PR[90,3] + 129.611;
   1:L PR[91] R[100]mm/sec CNT100;
   1:  PR[91,1] = PR[90,1] + 79.063;
   1:  PR[91,2] = PR[90,2] + 9.444;
   1:  PR[91,3] = PR[90,3] + 129.623;
   1:L PR[91] R[100]mm/sec CNT100;
   1:  PR[91,1] = PR[90,1] + 77.361;
   1:  PR[91,2] = PR[90,2] + 13.254;
   1:  PR[91,3] = PR[90,3] + 129.635;
   1:L PR[91] R[100]mm/sec CNT100;
   1:  PR[91,1] = PR[90,1] + 76.184;
   1:  PR[91,2] = PR[90,2] + 15.154;
   1:  PR[91,3] = PR[90,3] + 129.659;
   1:L PR[91] R[100]mm/sec CNT100;
   1:  PR[91,1] = PR[90,1] + 74.485;
   1:  PR[91,2] = PR[90,2] + 17.180;
   1:  PR[91,3] = PR[90,3] + 129.671;
   1:L PR[91] R[100]mm/sec CNT100;
   1:  PR[91,1] = PR[90,1] + 71.780;
   1:  PR[91,2] = PR[90,2] + 20.446;
   1:  PR[91,3] = PR[90,3] + 129.686;
   1:L PR[91] R[100]mm/sec CNT100;
   1:  PR[91,1] = PR[90,1] + 69.831;
   1:  PR[91,2] = PR[90,2] + 22.194;
   1:  PR[91,3] = PR[90,3] + 129.710;
   1:L PR[91] R[100]mm/sec CNT100;
   1:  PR[91,1] = PR[90,1] + 67.182;
   1:  PR[91,2] = PR[90,2] + 24.020;
   1:  PR[91,3] = PR[90,3] + 129.724;
   1:L PR[91] R[100]mm/sec CNT100;
   1:  PR[91,1] = PR[90,1] + 63.861;
   1:  PR[91,2] = PR[90,2] + 26.379;
   1:  PR[91,3] = PR[90,3] + 129.742;
   1:L PR[91] R[100]mm/sec CNT100;
   1:  PR[91,1] = PR[90,1] + 61.021;
   1:  PR[91,2] = PR[90,2] + 27.832;
   1:  PR[91,3] = PR[90,3] + 129.765;
   1:L PR[91] R[100]mm/sec CNT100;
   1:  PR[91,1] = PR[90,1] + 57.270;
   1:  PR[91,2] = PR[90,2] + 29.234;
   1:  PR[91,3] = PR[90,3] + 129.783;
   1:L PR[91] R[100]mm/sec CNT100;
   1:  PR[91,1] = PR[90,1] + 54.165;
   1:  PR[91,2] = PR[90,2] + 30.423;
   1:  PR[91,3] = PR[90,3] + 129.806;
   1:L PR[91] R[100]mm/sec CNT100;
   1:  PR[91,1] = PR[90,1] + 50.277;
   1:  PR[91,2] = PR[90,2] + 31.354;
   1:  PR[91,3] = PR[90,3] + 129.824;
   1:L PR[91] R[100]mm/sec CNT100;
   1:  PR[91,1] = PR[90,1] + 49.032;
   1:  PR[91,2] = PR[90,2] + 31.584;
   1:  PR[91,3] = PR[90,3] + 129.847;
   1:L PR[91] R[100]mm/sec CNT100;
   1:  PR[91,1] = PR[90,1] + 44.558;
   1:  PR[91,2] = PR[90,2] + 32.129;
   1:  PR[91,3] = PR[90,3] + 129.854;
   1:L PR[91] R[100]mm/sec CNT100;
   1:  PR[91,1] = PR[90,1] + 43.819;
   1:  PR[91,2] = PR[90,2] + 32.174;
   1:  PR[91,3] = PR[90,3] + 129.879;
   1:L PR[91] R[100]mm/sec CNT100;
   1:  PR[91,1] = PR[90,1] + 38.785;
   1:  PR[91,2] = PR[90,2] + 32.220;
   1:  PR[91,3] = PR[90,3] + 129.883;
   1:L PR[91] R[100]mm/sec CNT100;
   1:  PR[91,1] = PR[90,1] + 38.744;
   1:  PR[91,2] = PR[90,2] + 32.217;
   1:  PR[91,3] = PR[90,3] + 129.911;
   1:L PR[91] R[100]mm/sec CNT100;
   1:  PR[91,1] = PR[90,1] + 37.853;
   1:  PR[91,2] = PR[90,2] + 32.129;
   1:  PR[91,3] = PR[90,3] + 129.912;
   1:L PR[91] R[100]mm/sec CNT100;
   1:  PR[91,1] = PR[90,1] + 33.681;
   1:  PR[91,2] = PR[90,2] + 31.647;
   1:  PR[91,3] = PR[90,3] + 129.917;
   1:L PR[91] R[100]mm/sec CNT100;
   1:  PR[91,1] = PR[90,1] + 31.032;
   1:  PR[91,2] = PR[90,2] + 31.014;
   1:  PR[91,3] = PR[90,3] + 129.940;
   1:L PR[91] R[100]mm/sec CNT100;
   1:  PR[91,1] = PR[90,1] + 27.557;
   1:  PR[91,2] = PR[90,2] + 30.219;
   1:  PR[91,3] = PR[90,3] + 129.956;
   1:L PR[91] R[100]mm/sec CNT100;
   1:  PR[91,1] = PR[90,1] + 25.937;
   1:  PR[91,2] = PR[90,2] + 29.682;
   1:  PR[91,3] = PR[90,3] + 129.976;
   1:L PR[91] R[100]mm/sec CNT100;
   1:  PR[91,1] = PR[90,1] + 20.527;
   1:  PR[91,2] = PR[90,2] + 27.471;
   1:  PR[91,3] = PR[90,3] + 129.985;
   1:L PR[91] R[100]mm/sec CNT100;
   1:  PR[91,1] = PR[90,1] + 20.019;
   1:  PR[91,2] = PR[90,2] + 27.198;
   1:  PR[91,3] = PR[90,3] + 130.018;
   1:L PR[91] R[100]mm/sec CNT100;
   1:  PR[91,1] = PR[90,1] + 15.179;
   1:  PR[91,2] = PR[90,2] + 24.391;
   1:  PR[91,3] = PR[90,3] + 130.021;
   1:L PR[91] R[100]mm/sec CNT100;
   1:  PR[91,1] = PR[90,1] + 11.018;
   1:  PR[91,2] = PR[90,2] + 21.185;
   1:  PR[91,3] = PR[90,3] + 130.052;
   1:L PR[91] R[100]mm/sec CNT100;
   1:  PR[91,1] = PR[90,1] + 10.350;
   1:  PR[91,2] = PR[90,2] + 20.640;
   1:  PR[91,3] = PR[90,3] + 130.082;
   1:L PR[91] R[100]mm/sec CNT100;
   1:  PR[91,1] = PR[90,1] + 9.311;
   1:  PR[91,2] = PR[90,2] + 19.492;
   1:  PR[91,3] = PR[90,3] + 130.087;
   1:L PR[91] R[100]mm/sec CNT100;
   1:  PR[91,1] = PR[90,1] + 5.463;
   1:  PR[91,2] = PR[90,2] + 15.693;
   1:  PR[91,3] = PR[90,3] + 130.095;
   1:L PR[91] R[100]mm/sec CNT100;
   1:  PR[91,1] = PR[90,1] + 1.879;
   1:  PR[91,2] = PR[90,2] + 10.364;
   1:  PR[91,3] = PR[90,3] + 130.126;
   1:L PR[91] R[100]mm/sec CNT100;
   1:  PR[91,1] = PR[90,1] + -0.245;
   1:  PR[91,2] = PR[90,2] + 4.828;
   1:  PR[91,3] = PR[90,3] + 130.162;
   1:L PR[91] R[100]mm/sec CNT100;
   1:  PR[91] = PR[90];
   1:  PR[91,1] = PR[90,1] + 0.362;
   1:  PR[91,2] = PR[90,2] + 0.195;
   1:  PR[91,3] = PR[90,3] + 131.495;
   1:L PR[91] R[100]mm/sec CNT100;
   1:  PR[91,1] = PR[90,1] + 0.352;
   1:  PR[91,2] = PR[90,2] + -0.421;
   1:  PR[91,3] = PR[90,3] + 130.222;
   1:L PR[91] R[100]mm/sec CNT100;
   1:  PR[91,1] = PR[90,1] + 0.313;
   1:  PR[91,2] = PR[90,2] + -0.741;
   1:  PR[91,3] = PR[90,3] + 130.225;
   1:L PR[91] R[100]mm/sec CNT100;
   1:  PR[91,1] = PR[90,1] + 0.815;
   1:  PR[91,2] = PR[90,2] + -5.208;
   1:  PR[91,3] = PR[90,3] + 130.227;
   1:L PR[91] R[100]mm/sec CNT100;
   1:  PR[91,1] = PR[90,1] + 0.958;
   1:  PR[91,2] = PR[90,2] + -6.355;
   1:  PR[91,3] = PR[90,3] + 130.252;
   1:L PR[91] R[100]mm/sec CNT100;
   1:  PR[91,1] = PR[90,1] + 3.092;
   1:  PR[91,2] = PR[90,2] + -11.903;
   1:  PR[91,3] = PR[90,3] + 130.259;
   1:L PR[91] R[100]mm/sec CNT100;
   1:  PR[91,1] = PR[90,1] + 6.708;
   1:  PR[91,2] = PR[90,2] + -17.267;
   1:  PR[91,3] = PR[90,3] + 130.292;
   1:L PR[91] R[100]mm/sec CNT100;
   1:  PR[91,1] = PR[90,1] + 8.172;
   1:  PR[91,2] = PR[90,2] + -18.713;
   1:  PR[91,3] = PR[90,3] + 130.328;
   1:L PR[91] R[100]mm/sec CNT100;
   1:  PR[91,1] = PR[90,1] + 11.136;
   1:  PR[91,2] = PR[90,2] + -21.987;
   1:  PR[91,3] = PR[90,3] + 130.340;
   1:L PR[91] R[100]mm/sec CNT100;
   1:  PR[91,1] = PR[90,1] + 13.211;
   1:  PR[91,2] = PR[90,2] + -23.681;
   1:  PR[91,3] = PR[90,3] + 130.365;
   1:L PR[91] R[100]mm/sec CNT100;
   1:  PR[91,1] = PR[90,1] + 15.912;
   1:  PR[91,2] = PR[90,2] + -25.763;
   1:  PR[91,3] = PR[90,3] + 130.380;
   1:L PR[91] R[100]mm/sec CNT100;
   1:  PR[91,1] = PR[90,1] + 20.093;
   1:  PR[91,2] = PR[90,2] + -28.189;
   1:  PR[91,3] = PR[90,3] + 130.399;
   1:L PR[91] R[100]mm/sec CNT100;
   1:  PR[91,1] = PR[90,1] + 21.308;
   1:  PR[91,2] = PR[90,2] + -28.919;
   1:  PR[91,3] = PR[90,3] + 130.426;
   1:L PR[91] R[100]mm/sec CNT100;
   1:  PR[91,1] = PR[90,1] + 21.724;
   1:  PR[91,2] = PR[90,2] + -29.109;
   1:  PR[91,3] = PR[90,3] + 130.434;
   1:L PR[91] R[100]mm/sec CNT100;
   1:  PR[91,1] = PR[90,1] + 26.424;
   1:  PR[91,2] = PR[90,2] + -31.039;
   1:  PR[91,3] = PR[90,3] + 130.437;
   1:L PR[91] R[100]mm/sec CNT100;
   1:  PR[91,1] = PR[90,1] + 28.798;
   1:  PR[91,2] = PR[90,2] + -31.826;
   1:  PR[91,3] = PR[90,3] + 130.465;
   1:L PR[91] R[100]mm/sec CNT100;
   1:  PR[91,1] = PR[90,1] + 30.884;
   1:  PR[91,2] = PR[90,2] + -32.335;
   1:  PR[91,3] = PR[90,3] + 130.479;
   1:L PR[91] R[100]mm/sec CNT100;
   1:  PR[91,1] = PR[90,1] + 34.572;
   1:  PR[91,2] = PR[90,2] + -33.156;
   1:  PR[91,3] = PR[90,3] + 130.491;
   1:L PR[91] R[100]mm/sec CNT100;
   1:  PR[91,1] = PR[90,1] + 35.925;
   1:  PR[91,2] = PR[90,2] + -33.313;
   1:  PR[91,3] = PR[90,3] + 130.513;
   1:L PR[91] R[100]mm/sec CNT100;
   1:  PR[91,1] = PR[90,1] + 39.369;
   1:  PR[91,2] = PR[90,2] + -33.655;
   1:  PR[91,3] = PR[90,3] + 130.520;
   1:L PR[91] R[100]mm/sec CNT100;
   1:  PR[91,1] = PR[90,1] + 39.812;
   1:  PR[91,2] = PR[90,2] + -33.682;
   1:  PR[91,3] = PR[90,3] + 130.540;
   1:L PR[91] R[100]mm/sec CNT100;
   1:  PR[91,1] = PR[90,1] + 44.502;
   1:  PR[91,2] = PR[90,2] + -33.639;
   1:  PR[91,3] = PR[90,3] + 130.542;
   1:L PR[91] R[100]mm/sec CNT100;
   1:  PR[91,1] = PR[90,1] + 45.596;
   1:  PR[91,2] = PR[90,2] + -33.572;
   1:  PR[91,3] = PR[90,3] + 130.568;
   1:L PR[91] R[100]mm/sec CNT100;
   1:  PR[91,1] = PR[90,1] + 49.763;
   1:  PR[91,2] = PR[90,2] + -33.065;
   1:  PR[91,3] = PR[90,3] + 130.575;
   1:L PR[91] R[100]mm/sec CNT100;
   1:  PR[91,1] = PR[90,1] + 51.316;
   1:  PR[91,2] = PR[90,2] + -32.778;
   1:  PR[91,3] = PR[90,3] + 130.598;
   1:L PR[91] R[100]mm/sec CNT100;
   1:  PR[91,1] = PR[90,1] + 54.941;
   1:  PR[91,2] = PR[90,2] + -31.910;
   1:  PR[91,3] = PR[90,3] + 130.607;
   1:L PR[91] R[100]mm/sec CNT100;
   1:  PR[91,1] = PR[90,1] + 57.844;
   1:  PR[91,2] = PR[90,2] + -30.829;
   1:  PR[91,3] = PR[90,3] + 130.628;
   1:L PR[91] R[100]mm/sec CNT100;
   1:  PR[91,1] = PR[90,1] + 62.031;
   1:  PR[91,2] = PR[90,2] + -29.226;
   1:  PR[91,3] = PR[90,3] + 130.645;
   1:L PR[91] R[100]mm/sec CNT100;
   1:  PR[91,1] = PR[90,1] + 64.687;
   1:  PR[91,2] = PR[90,2] + -27.868;
   1:  PR[91,3] = PR[90,3] + 130.671;
   1:L PR[91] R[100]mm/sec CNT100;
   1:  PR[91,1] = PR[90,1] + 66.842;
   1:  PR[91,2] = PR[90,2] + -26.388;
   1:  PR[91,3] = PR[90,3] + 130.687;
   1:L PR[91] R[100]mm/sec CNT100;
   1:  PR[91,1] = PR[90,1] + 70.792;
   1:  PR[91,2] = PR[90,2] + -23.581;
   1:  PR[91,3] = PR[90,3] + 130.702;
   1:L PR[91] R[100]mm/sec CNT100;
   1:  PR[91,1] = PR[90,1] + 72.613;
   1:  PR[91,2] = PR[90,2] + -21.948;
   1:  PR[91,3] = PR[90,3] + 130.729;
   1:L PR[91] R[100]mm/sec CNT100;
   1:  PR[91,1] = PR[90,1] + 74.064;
   1:  PR[91,2] = PR[90,2] + -20.220;
   1:  PR[91,3] = PR[90,3] + 130.743;
   1:L PR[91] R[100]mm/sec CNT100;
   1:  PR[91,1] = PR[90,1] + 77.104;
   1:  PR[91,2] = PR[90,2] + -16.548;
   1:  PR[91,3] = PR[90,3] + 130.756;
   1:L PR[91] R[100]mm/sec CNT100;
   1:  PR[91,1] = PR[90,1] + 78.187;
   1:  PR[91,2] = PR[90,2] + -14.801;
   1:  PR[91,3] = PR[90,3] + 130.782;
   1:L PR[91] R[100]mm/sec CNT100;
   1:  PR[91,1] = PR[90,1] + 78.986;
   1:  PR[91,2] = PR[90,2] + -12.913;
   1:  PR[91,3] = PR[90,3] + 130.794;
   1:L PR[91] R[100]mm/sec CNT100;
   1:  PR[91,1] = PR[90,1] + 80.840;
   1:  PR[91,2] = PR[90,2] + -8.763;
   1:  PR[91,3] = PR[90,3] + 130.806;
   1:L PR[91] R[100]mm/sec CNT100;
   1:  PR[91,1] = PR[90,1] + 81.278;
   1:  PR[91,2] = PR[90,2] + -6.999;
   1:  PR[91,3] = PR[90,3] + 130.831;
   1:L PR[91] R[100]mm/sec CNT100;
   1:  PR[91,1] = PR[90,1] + 81.441;
   1:  PR[91,2] = PR[90,2] + -4.995;
   1:  PR[91,3] = PR[90,3] + 130.841;
   1:L PR[91] R[100]mm/sec CNT100;
   1:  PR[91,1] = PR[90,1] + 82.054;
   1:  PR[91,2] = PR[90,2] + -0.670;
   1:  PR[91,3] = PR[90,3] + 130.853;
   1:L PR[91] R[100]mm/sec CNT100;
   1:  PR[91,1] = PR[90,1] + 81.904;
   1:  PR[91,2] = PR[90,2] + 1.172;
   1:  PR[91,3] = PR[90,3] + 130.877;
   1:L PR[91] R[100]mm/sec CNT100;
   1:  PR[91,1] = PR[90,1] + 81.292;
   1:  PR[91,2] = PR[90,2] + 5.483;
   1:  PR[91,3] = PR[90,3] + 130.888;
   1:L PR[91] R[100]mm/sec CNT100;
   1:  PR[91,1] = PR[90,1] + 80.835;
   1:  PR[91,2] = PR[90,2] + 7.323;
   1:  PR[91,3] = PR[90,3] + 130.912;
   1:L PR[91] R[100]mm/sec CNT100;
   1:  PR[91,1] = PR[90,1] + 80.016;
   1:  PR[91,2] = PR[90,2] + 9.254;
   1:  PR[91,3] = PR[90,3] + 130.923;
   1:L PR[91] R[100]mm/sec CNT100;
   1:  PR[91,1] = PR[90,1] + 78.197;
   1:  PR[91,2] = PR[90,2] + 13.327;
   1:  PR[91,3] = PR[90,3] + 130.934;
   1:L PR[91] R[100]mm/sec CNT100;
   1:  PR[91,1] = PR[90,1] + 77.108;
   1:  PR[91,2] = PR[90,2] + 15.084;
   1:  PR[91,3] = PR[90,3] + 130.959;
   1:L PR[91] R[100]mm/sec CNT100;
   1:  PR[91,1] = PR[90,1] + 75.528;
   1:  PR[91,2] = PR[90,2] + 16.967;
   1:  PR[91,3] = PR[90,3] + 130.971;
   1:L PR[91] R[100]mm/sec CNT100;
   1:  PR[91,1] = PR[90,1] + 72.607;
   1:  PR[91,2] = PR[90,2] + 20.495;
   1:  PR[91,3] = PR[90,3] + 130.985;
   1:L PR[91] R[100]mm/sec CNT100;
   1:  PR[91,1] = PR[90,1] + 70.802;
   1:  PR[91,2] = PR[90,2] + 22.113;
   1:  PR[91,3] = PR[90,3] + 131.011;
   1:L PR[91] R[100]mm/sec CNT100;
   1:  PR[91,1] = PR[90,1] + 68.336;
   1:  PR[91,2] = PR[90,2] + 23.814;
   1:  PR[91,3] = PR[90,3] + 131.024;
   1:L PR[91] R[100]mm/sec CNT100;
   1:  PR[91,1] = PR[90,1] + 64.672;
   1:  PR[91,2] = PR[90,2] + 26.417;
   1:  PR[91,3] = PR[90,3] + 131.041;
   1:L PR[91] R[100]mm/sec CNT100;
   1:  PR[91,1] = PR[90,1] + 62.037;
   1:  PR[91,2] = PR[90,2] + 27.764;
   1:  PR[91,3] = PR[90,3] + 131.066;
   1:L PR[91] R[100]mm/sec CNT100;
   1:  PR[91,1] = PR[90,1] + 58.543;
   1:  PR[91,2] = PR[90,2] + 29.071;
   1:  PR[91,3] = PR[90,3] + 131.083;
   1:L PR[91] R[100]mm/sec CNT100;
   1:  PR[91,1] = PR[90,1] + 54.931;
   1:  PR[91,2] = PR[90,2] + 30.453;
   1:  PR[91,3] = PR[90,3] + 131.104;
   1:L PR[91] R[100]mm/sec CNT100;
   1:  PR[91,1] = PR[90,1] + 51.315;
   1:  PR[91,2] = PR[90,2] + 31.319;
   1:  PR[91,3] = PR[90,3] + 131.126;
   1:L PR[91] R[100]mm/sec CNT100;
   1:  PR[91,1] = PR[90,1] + 49.762;
   1:  PR[91,2] = PR[90,2] + 31.606;
   1:  PR[91,3] = PR[90,3] + 131.147;
   1:L PR[91] R[100]mm/sec CNT100;
   1:  PR[91,1] = PR[90,1] + 45.595;
   1:  PR[91,2] = PR[90,2] + 32.114;
   1:  PR[91,3] = PR[90,3] + 131.155;
   1:L PR[91] R[100]mm/sec CNT100;
   1:  PR[91,1] = PR[90,1] + 44.501;
   1:  PR[91,2] = PR[90,2] + 32.180;
   1:  PR[91,3] = PR[90,3] + 131.179;
   1:L PR[91] R[100]mm/sec CNT100;
   1:  PR[91,1] = PR[90,1] + 39.812;
   1:  PR[91,2] = PR[90,2] + 32.223;
   1:  PR[91,3] = PR[90,3] + 131.185;
   1:L PR[91] R[100]mm/sec CNT100;
   1:  PR[91,1] = PR[90,1] + 39.369;
   1:  PR[91,2] = PR[90,2] + 32.196;
   1:  PR[91,3] = PR[90,3] + 131.212;
   1:L PR[91] R[100]mm/sec CNT100;
   1:  PR[91,1] = PR[90,1] + 35.925;
   1:  PR[91,2] = PR[90,2] + 31.854;
   1:  PR[91,3] = PR[90,3] + 131.214;
   1:L PR[91] R[100]mm/sec CNT100;
   1:  PR[91,1] = PR[90,1] + 34.580;
   1:  PR[91,2] = PR[90,2] + 31.699;
   1:  PR[91,3] = PR[90,3] + 131.233;
   1:L PR[91] R[100]mm/sec CNT100;
   1:  PR[91,1] = PR[90,1] + 28.790;
   1:  PR[91,2] = PR[90,2] + 30.364;
   1:  PR[91,3] = PR[90,3] + 131.241;
   1:L PR[91] R[100]mm/sec CNT100;
   1:  PR[91,1] = PR[90,1] + 26.427;
   1:  PR[91,2] = PR[90,2] + 29.581;
   1:  PR[91,3] = PR[90,3] + 131.274;
   1:L PR[91] R[100]mm/sec CNT100;
   1:  PR[91,1] = PR[90,1] + 21.732;
   1:  PR[91,2] = PR[90,2] + 27.653;
   1:  PR[91,3] = PR[90,3] + 131.288;
   1:L PR[91] R[100]mm/sec CNT100;
   1:  PR[91,1] = PR[90,1] + 21.314;
   1:  PR[91,2] = PR[90,2] + 27.463;
   1:  PR[91,3] = PR[90,3] + 131.317;
   1:L PR[91] R[100]mm/sec CNT100;
   1:  PR[91,1] = PR[90,1] + 20.093;
   1:  PR[91,2] = PR[90,2] + 26.730;
   1:  PR[91,3] = PR[90,3] + 131.320;
   1:L PR[91] R[100]mm/sec CNT100;
   1:  PR[91,1] = PR[90,1] + 15.918;
   1:  PR[91,2] = PR[90,2] + 24.308;
   1:  PR[91,3] = PR[90,3] + 131.328;
   1:L PR[91] R[100]mm/sec CNT100;
   1:  PR[91,1] = PR[90,1] + 13.220;
   1:  PR[91,2] = PR[90,2] + 22.229;
   1:  PR[91,3] = PR[90,3] + 131.355;
   1:L PR[91] R[100]mm/sec CNT100;
   1:  PR[91,1] = PR[90,1] + 11.141;
   1:  PR[91,2] = PR[90,2] + 20.533;
   1:  PR[91,3] = PR[90,3] + 131.374;
   1:L PR[91] R[100]mm/sec CNT100;
   1:  PR[91,1] = PR[90,1] + 8.172;
   1:  PR[91,2] = PR[90,2] + 17.254;
   1:  PR[91,3] = PR[90,3] + 131.389;
   1:L PR[91] R[100]mm/sec CNT100;
   1:  PR[91,1] = PR[90,1] + 6.712;
   1:  PR[91,2] = PR[90,2] + 15.813;
   1:  PR[91,3] = PR[90,3] + 131.414;
   1:L PR[91] R[100]mm/sec CNT100;
   1:  PR[91,1] = PR[90,1] + 3.093;
   1:  PR[91,2] = PR[90,2] + 10.446;
   1:  PR[91,3] = PR[90,3] + 131.425;
   1:L PR[91] R[100]mm/sec CNT100;
   1:  PR[91,1] = PR[90,1] + 0.957;
   1:  PR[91,2] = PR[90,2] + 4.895;
   1:  PR[91,3] = PR[90,3] + 131.462;
   1:L PR[91] R[100]mm/sec CNT100;
   1:  PR[91] = PR[90];
   1:  PR[91,1] = PR[90,1] + 1.748;
   1:  PR[91,2] = PR[90,2] + 1.763;
   1:  PR[91,3] = PR[90,3] + 132.795;
   1:L PR[91] R[100]mm/sec CNT100;
   1:  PR[91,1] = PR[90,1] + 1.741;
   1:  PR[91,2] = PR[90,2] + 1.333;
   1:  PR[91,3] = PR[90,3] + 131.513;
   1:L PR[91] R[100]mm/sec CNT100;
   1:  PR[91,1] = PR[90,1] + 1.484;
   1:  PR[91,2] = PR[90,2] + -0.741;
   1:  PR[91,3] = PR[90,3] + 131.515;
   1:L PR[91] R[100]mm/sec CNT100;
   1:  PR[91,1] = PR[90,1] + 1.837;
   1:  PR[91,2] = PR[90,2] + -3.875;
   1:  PR[91,3] = PR[90,3] + 131.527;
   1:L PR[91] R[100]mm/sec CNT100;
   1:  PR[91,1] = PR[90,1] + 2.150;
   1:  PR[91,2] = PR[90,2] + -6.396;
   1:  PR[91,3] = PR[90,3] + 131.545;
   1:L PR[91] R[100]mm/sec CNT100;
   1:  PR[91,1] = PR[90,1] + 4.306;
   1:  PR[91,2] = PR[90,2] + -11.984;
   1:  PR[91,3] = PR[90,3] + 131.559;
   1:L PR[91] R[100]mm/sec CNT100;
   1:  PR[91,1] = PR[90,1] + 7.274;
   1:  PR[91,2] = PR[90,2] + -16.379;
   1:  PR[91,3] = PR[90,3] + 131.593;
   1:L PR[91] R[100]mm/sec CNT100;
   1:  PR[91,1] = PR[90,1] + 7.897;
   1:  PR[91,2] = PR[90,2] + -17.413;
   1:  PR[91,3] = PR[90,3] + 131.623;
   1:L PR[91] R[100]mm/sec CNT100;
   1:  PR[91,1] = PR[90,1] + 8.179;
   1:  PR[91,2] = PR[90,2] + -17.740;
   1:  PR[91,3] = PR[90,3] + 131.630;
   1:L PR[91] R[100]mm/sec CNT100;
   1:  PR[91,1] = PR[90,1] + 11.928;
   1:  PR[91,2] = PR[90,2] + -21.881;
   1:  PR[91,3] = PR[90,3] + 131.632;
   1:L PR[91] R[100]mm/sec CNT100;
   1:  PR[91,1] = PR[90,1] + 15.413;
   1:  PR[91,2] = PR[90,2] + -24.726;
   1:  PR[91,3] = PR[90,3] + 131.663;
   1:L PR[91] R[100]mm/sec CNT100;
   1:  PR[91,1] = PR[90,1] + 16.652;
   1:  PR[91,2] = PR[90,2] + -25.681;
   1:  PR[91,3] = PR[90,3] + 131.689;
   1:L PR[91] R[100]mm/sec CNT100;
   1:  PR[91,1] = PR[90,1] + 18.618;
   1:  PR[91,2] = PR[90,2] + -26.821;
   1:  PR[91,3] = PR[90,3] + 131.698;
   1:L PR[91] R[100]mm/sec CNT100;
   1:  PR[91,1] = PR[90,1] + 22.026;
   1:  PR[91,2] = PR[90,2] + -28.868;
   1:  PR[91,3] = PR[90,3] + 131.710;
   1:L PR[91] R[100]mm/sec CNT100;
   1:  PR[91,1] = PR[90,1] + 23.376;
   1:  PR[91,2] = PR[90,2] + -29.485;
   1:  PR[91,3] = PR[90,3] + 131.733;
   1:L PR[91] R[100]mm/sec CNT100;
   1:  PR[91,1] = PR[90,1] + 26.914;
   1:  PR[91,2] = PR[90,2] + -30.938;
   1:  PR[91,3] = PR[90,3] + 131.741;
   1:L PR[91] R[100]mm/sec CNT100;
   1:  PR[91,1] = PR[90,1] + 30.032;
   1:  PR[91,2] = PR[90,2] + -31.971;
   1:  PR[91,3] = PR[90,3] + 131.763;
   1:L PR[91] R[100]mm/sec CNT100;
   1:  PR[91,1] = PR[90,1] + 31.193;
   1:  PR[91,2] = PR[90,2] + -32.255;
   1:  PR[91,3] = PR[90,3] + 131.781;
   1:L PR[91] R[100]mm/sec CNT100;
   1:  PR[91,1] = PR[90,1] + 34.201;
   1:  PR[91,2] = PR[90,2] + -32.924;
   1:  PR[91,3] = PR[90,3] + 131.788;
   1:L PR[91] R[100]mm/sec CNT100;
   1:  PR[91,1] = PR[90,1] + 35.483;
   1:  PR[91,2] = PR[90,2] + -33.185;
   1:  PR[91,3] = PR[90,3] + 131.805;
   1:L PR[91] R[100]mm/sec CNT100;
   1:  PR[91,1] = PR[90,1] + 39.994;
   1:  PR[91,2] = PR[90,2] + -33.633;
   1:  PR[91,3] = PR[90,3] + 131.812;
   1:L PR[91] R[100]mm/sec CNT100;
   1:  PR[91,1] = PR[90,1] + 40.839;
   1:  PR[91,2] = PR[90,2] + -33.685;
   1:  PR[91,3] = PR[90,3] + 131.838;
   1:L PR[91] R[100]mm/sec CNT100;
   1:  PR[91,1] = PR[90,1] + 45.184;
   1:  PR[91,2] = PR[90,2] + -33.646;
   1:  PR[91,3] = PR[90,3] + 131.843;
   1:L PR[91] R[100]mm/sec CNT100;
   1:  PR[91,1] = PR[90,1] + 46.633;
   1:  PR[91,2] = PR[90,2] + -33.557;
   1:  PR[91,3] = PR[90,3] + 131.867;
   1:L PR[91] R[100]mm/sec CNT100;
   1:  PR[91,1] = PR[90,1] + 50.493;
   1:  PR[91,2] = PR[90,2] + -33.087;
   1:  PR[91,3] = PR[90,3] + 131.875;
   1:L PR[91] R[100]mm/sec CNT100;
   1:  PR[91,1] = PR[90,1] + 52.355;
   1:  PR[91,2] = PR[90,2] + -32.743;
   1:  PR[91,3] = PR[90,3] + 131.897;
   1:L PR[91] R[100]mm/sec CNT100;
   1:  PR[91,1] = PR[90,1] + 55.708;
   1:  PR[91,2] = PR[90,2] + -31.940;
   1:  PR[91,3] = PR[90,3] + 131.908;
   1:L PR[91] R[100]mm/sec CNT100;
   1:  PR[91,1] = PR[90,1] + 58.394;
   1:  PR[91,2] = PR[90,2] + -30.940;
   1:  PR[91,3] = PR[90,3] + 131.927;
   1:L PR[91] R[100]mm/sec CNT100;
   1:  PR[91,1] = PR[90,1] + 63.047;
   1:  PR[91,2] = PR[90,2] + -29.159;
   1:  PR[91,3] = PR[90,3] + 131.943;
   1:L PR[91] R[100]mm/sec CNT100;
   1:  PR[91,1] = PR[90,1] + 65.497;
   1:  PR[91,2] = PR[90,2] + -27.905;
   1:  PR[91,3] = PR[90,3] + 131.971;
   1:L PR[91] R[100]mm/sec CNT100;
   1:  PR[91,1] = PR[90,1] + 67.489;
   1:  PR[91,2] = PR[90,2] + -26.537;
   1:  PR[91,3] = PR[90,3] + 131.987;
   1:L PR[91] R[100]mm/sec CNT100;
   1:  PR[91,1] = PR[90,1] + 71.764;
   1:  PR[91,2] = PR[90,2] + -23.500;
   1:  PR[91,3] = PR[90,3] + 132.001;
   1:L PR[91] R[100]mm/sec CNT100;
   1:  PR[91,1] = PR[90,1] + 73.440;
   1:  PR[91,2] = PR[90,2] + -21.997;
   1:  PR[91,3] = PR[90,3] + 132.030;
   1:L PR[91] R[100]mm/sec CNT100;
   1:  PR[91,1] = PR[90,1] + 74.781;
   1:  PR[91,2] = PR[90,2] + -20.400;
   1:  PR[91,3] = PR[90,3] + 132.043;
   1:L PR[91] R[100]mm/sec CNT100;
   1:  PR[91,1] = PR[90,1] + 78.028;
   1:  PR[91,2] = PR[90,2] + -16.478;
   1:  PR[91,3] = PR[90,3] + 132.054;
   1:L PR[91] R[100]mm/sec CNT100;
   1:  PR[91,1] = PR[90,1] + 79.023;
   1:  PR[91,2] = PR[90,2] + -14.874;
   1:  PR[91,3] = PR[90,3] + 132.083;
   1:L PR[91] R[100]mm/sec CNT100;
   1:  PR[91,1] = PR[90,1] + 79.761;
   1:  PR[91,2] = PR[90,2] + -13.129;
   1:  PR[91,3] = PR[90,3] + 132.094;
   1:L PR[91] R[100]mm/sec CNT100;
   1:  PR[91,1] = PR[90,1] + 81.729;
   1:  PR[91,2] = PR[90,2] + -8.722;
   1:  PR[91,3] = PR[90,3] + 132.104;
   1:L PR[91] R[100]mm/sec CNT100;
   1:  PR[91,1] = PR[90,1] + 82.130;
   1:  PR[91,2] = PR[90,2] + -7.109;
   1:  PR[91,3] = PR[90,3] + 132.132;
   1:L PR[91] R[100]mm/sec CNT100;
   1:  PR[91,1] = PR[90,1] + 82.281;
   1:  PR[91,2] = PR[90,2] + -5.255;
   1:  PR[91,3] = PR[90,3] + 132.141;
   1:L PR[91] R[100]mm/sec CNT100;
   1:  PR[91,1] = PR[90,1] + 82.931;
   1:  PR[91,2] = PR[90,2] + -0.670;
   1:  PR[91,3] = PR[90,3] + 132.151;
   1:L PR[91] R[100]mm/sec CNT100;
   1:  PR[91,1] = PR[90,1] + 82.793;
   1:  PR[91,2] = PR[90,2] + 1.020;
   1:  PR[91,3] = PR[90,3] + 132.177;
   1:L PR[91] R[100]mm/sec CNT100;
   1:  PR[91,1] = PR[90,1] + 82.145;
   1:  PR[91,2] = PR[90,2] + 5.592;
   1:  PR[91,3] = PR[90,3] + 132.187;
   1:L PR[91] R[100]mm/sec CNT100;
   1:  PR[91,1] = PR[90,1] + 81.724;
   1:  PR[91,2] = PR[90,2] + 7.283;
   1:  PR[91,3] = PR[90,3] + 132.213;
   1:L PR[91] R[100]mm/sec CNT100;
   1:  PR[91,1] = PR[90,1] + 80.969;
   1:  PR[91,2] = PR[90,2] + 9.063;
   1:  PR[91,3] = PR[90,3] + 132.223;
   1:L PR[91] R[100]mm/sec CNT100;
   1:  PR[91,1] = PR[90,1] + 79.032;
   1:  PR[91,2] = PR[90,2] + 13.399;
   1:  PR[91,3] = PR[90,3] + 132.234;
   1:L PR[91] R[100]mm/sec CNT100;
   1:  PR[91,1] = PR[90,1] + 78.032;
   1:  PR[91,2] = PR[90,2] + 15.014;
   1:  PR[91,3] = PR[90,3] + 132.260;
   1:L PR[91] R[100]mm/sec CNT100;
   1:  PR[91,1] = PR[90,1] + 76.572;
   1:  PR[91,2] = PR[90,2] + 16.755;
   1:  PR[91,3] = PR[90,3] + 132.271;
   1:L PR[91] R[100]mm/sec CNT100;
   1:  PR[91,1] = PR[90,1] + 73.434;
   1:  PR[91,2] = PR[90,2] + 20.543;
   1:  PR[91,3] = PR[90,3] + 132.284;
   1:L PR[91] R[100]mm/sec CNT100;
   1:  PR[91,1] = PR[90,1] + 71.773;
   1:  PR[91,2] = PR[90,2] + 22.033;
   1:  PR[91,3] = PR[90,3] + 132.312;
   1:L PR[91] R[100]mm/sec CNT100;
   1:  PR[91,1] = PR[90,1] + 69.490;
   1:  PR[91,2] = PR[90,2] + 23.607;
   1:  PR[91,3] = PR[90,3] + 132.324;
   1:L PR[91] R[100]mm/sec CNT100;
   1:  PR[91,1] = PR[90,1] + 65.482;
   1:  PR[91,2] = PR[90,2] + 26.454;
   1:  PR[91,3] = PR[90,3] + 132.340;
   1:L PR[91] R[100]mm/sec CNT100;
   1:  PR[91,1] = PR[90,1] + 63.052;
   1:  PR[91,2] = PR[90,2] + 27.697;
   1:  PR[91,3] = PR[90,3] + 132.367;
   1:L PR[91] R[100]mm/sec CNT100;
   1:  PR[91,1] = PR[90,1] + 59.815;
   1:  PR[91,2] = PR[90,2] + 28.907;
   1:  PR[91,3] = PR[90,3] + 132.383;
   1:L PR[91] R[100]mm/sec CNT100;
   1:  PR[91,1] = PR[90,1] + 55.697;
   1:  PR[91,2] = PR[90,2] + 30.484;
   1:  PR[91,3] = PR[90,3] + 132.402;
   1:L PR[91] R[100]mm/sec CNT100;
   1:  PR[91,1] = PR[90,1] + 52.353;
   1:  PR[91,2] = PR[90,2] + 31.285;
   1:  PR[91,3] = PR[90,3] + 132.427;
   1:L PR[91] R[100]mm/sec CNT100;
   1:  PR[91,1] = PR[90,1] + 50.491;
   1:  PR[91,2] = PR[90,2] + 31.628;
   1:  PR[91,3] = PR[90,3] + 132.446;
   1:L PR[91] R[100]mm/sec CNT100;
   1:  PR[91,1] = PR[90,1] + 46.631;
   1:  PR[91,2] = PR[90,2] + 32.098;
   1:  PR[91,3] = PR[90,3] + 132.457;
   1:L PR[91] R[100]mm/sec CNT100;
   1:  PR[91,1] = PR[90,1] + 45.183;
   1:  PR[91,2] = PR[90,2] + 32.187;
   1:  PR[91,3] = PR[90,3] + 132.479;
   1:L PR[91] R[100]mm/sec CNT100;
   1:  PR[91,1] = PR[90,1] + 40.838;
   1:  PR[91,2] = PR[90,2] + 32.226;
   1:  PR[91,3] = PR[90,3] + 132.487;
   1:L PR[91] R[100]mm/sec CNT100;
   1:  PR[91,1] = PR[90,1] + 39.993;
   1:  PR[91,2] = PR[90,2] + 32.175;
   1:  PR[91,3] = PR[90,3] + 132.511;
   1:L PR[91] R[100]mm/sec CNT100;
   1:  PR[91,1] = PR[90,1] + 35.483;
   1:  PR[91,2] = PR[90,2] + 31.727;
   1:  PR[91,3] = PR[90,3] + 132.516;
   1:L PR[91] R[100]mm/sec CNT100;
   1:  PR[91,1] = PR[90,1] + 34.207;
   1:  PR[91,2] = PR[90,2] + 31.467;
   1:  PR[91,3] = PR[90,3] + 132.542;
   1:L PR[91] R[100]mm/sec CNT100;
   1:  PR[91,1] = PR[90,1] + 30.021;
   1:  PR[91,2] = PR[90,2] + 30.508;
   1:  PR[91,3] = PR[90,3] + 132.549;
   1:L PR[91] R[100]mm/sec CNT100;
   1:  PR[91,1] = PR[90,1] + 26.916;
   1:  PR[91,2] = PR[90,2] + 29.480;
   1:  PR[91,3] = PR[90,3] + 132.573;
   1:L PR[91] R[100]mm/sec CNT100;
   1:  PR[91,1] = PR[90,1] + 23.382;
   1:  PR[91,2] = PR[90,2] + 28.029;
   1:  PR[91,3] = PR[90,3] + 132.592;
   1:L PR[91] R[100]mm/sec CNT100;
   1:  PR[91,1] = PR[90,1] + 22.031;
   1:  PR[91,2] = PR[90,2] + 27.412;
   1:  PR[91,3] = PR[90,3] + 132.613;
   1:L PR[91] R[100]mm/sec CNT100;
   1:  PR[91,1] = PR[90,1] + 18.617;
   1:  PR[91,2] = PR[90,2] + 25.363;
   1:  PR[91,3] = PR[90,3] + 132.621;
   1:L PR[91] R[100]mm/sec CNT100;
   1:  PR[91,1] = PR[90,1] + 16.657;
   1:  PR[91,2] = PR[90,2] + 24.226;
   1:  PR[91,3] = PR[90,3] + 132.644;
   1:L PR[91] R[100]mm/sec CNT100;
   1:  PR[91,1] = PR[90,1] + 15.421;
   1:  PR[91,2] = PR[90,2] + 23.273;
   1:  PR[91,3] = PR[90,3] + 132.657;
   1:L PR[91] R[100]mm/sec CNT100;
   1:  PR[91,1] = PR[90,1] + 11.932;
   1:  PR[91,2] = PR[90,2] + 20.427;
   1:  PR[91,3] = PR[90,3] + 132.665;
   1:L PR[91] R[100]mm/sec CNT100;
   1:  PR[91,1] = PR[90,1] + 8.185;
   1:  PR[91,2] = PR[90,2] + 16.288;
   1:  PR[91,3] = PR[90,3] + 132.691;
   1:L PR[91] R[100]mm/sec CNT100;
   1:  PR[91,1] = PR[90,1] + 7.900;
   1:  PR[91,2] = PR[90,2] + 15.958;
   1:  PR[91,3] = PR[90,3] + 132.722;
   1:L PR[91] R[100]mm/sec CNT100;
   1:  PR[91,1] = PR[90,1] + 7.273;
   1:  PR[91,2] = PR[90,2] + 14.919;
   1:  PR[91,3] = PR[90,3] + 132.725;
   1:L PR[91] R[100]mm/sec CNT100;
   1:  PR[91,1] = PR[90,1] + 4.307;
   1:  PR[91,2] = PR[90,2] + 10.528;
   1:  PR[91,3] = PR[90,3] + 132.731;
   1:L PR[91] R[100]mm/sec CNT100;
   1:  PR[91,1] = PR[90,1] + 2.150;
   1:  PR[91,2] = PR[90,2] + 4.936;
   1:  PR[91,3] = PR[90,3] + 132.761;
   1:L PR[91] R[100]mm/sec CNT100;
   1:  PR[91] = PR[90];
   1:  PR[91,1] = PR[90,1] + 3.133;
   1:  PR[91,2] = PR[90,2] + 3.330;
   1:  PR[91,3] = PR[90,3] + 134.095;
   1:L PR[91] R[100]mm/sec CNT100;
   1:  PR[91,1] = PR[90,1] + 3.130;
   1:  PR[91,2] = PR[90,2] + 3.088;
   1:  PR[91,3] = PR[90,3] + 132.804;
   1:L PR[91] R[100]mm/sec CNT100;
   1:  PR[91,1] = PR[90,1] + 2.655;
   1:  PR[91,2] = PR[90,2] + -0.741;
   1:  PR[91,3] = PR[90,3] + 132.806;
   1:L PR[91] R[100]mm/sec CNT100;
   1:  PR[91,1] = PR[90,1] + 2.858;
   1:  PR[91,2] = PR[90,2] + -2.541;
   1:  PR[91,3] = PR[90,3] + 132.827;
   1:L PR[91] R[100]mm/sec CNT100;
   1:  PR[91,1] = PR[90,1] + 3.342;
   1:  PR[91,2] = PR[90,2] + -6.438;
   1:  PR[91,3] = PR[90,3] + 132.838;
   1:L PR[91] R[100]mm/sec CNT100;
   1:  PR[91,1] = PR[90,1] + 5.520;
   1:  PR[91,2] = PR[90,2] + -12.066;
   1:  PR[91,3] = PR[90,3] + 132.860;
   1:L PR[91] R[100]mm/sec CNT100;
   1:  PR[91,1] = PR[90,1] + 6.134;
   1:  PR[91,2] = PR[90,2] + -12.975;
   1:  PR[91,3] = PR[90,3] + 132.894;
   1:L PR[91] R[100]mm/sec CNT100;
   1:  PR[91,1] = PR[90,1] + 8.743;
   1:  PR[91,2] = PR[90,2] + -17.303;
   1:  PR[91,3] = PR[90,3] + 132.900;
   1:L PR[91] R[100]mm/sec CNT100;
   1:  PR[91,1] = PR[90,1] + 10.213;
   1:  PR[91,2] = PR[90,2] + -19.006;
   1:  PR[91,3] = PR[90,3] + 132.928;
   1:L PR[91] R[100]mm/sec CNT100;
   1:  PR[91,1] = PR[90,1] + 12.719;
   1:  PR[91,2] = PR[90,2] + -21.775;
   1:  PR[91,3] = PR[90,3] + 132.941;
   1:L PR[91] R[100]mm/sec CNT100;
   1:  PR[91,1] = PR[90,1] + 17.442;
   1:  PR[91,2] = PR[90,2] + -25.633;
   1:  PR[91,3] = PR[90,3] + 132.962;
   1:L PR[91] R[100]mm/sec CNT100;
   1:  PR[91,1] = PR[90,1] + 21.510;
   1:  PR[91,2] = PR[90,2] + -28.062;
   1:  PR[91,3] = PR[90,3] + 132.997;
   1:L PR[91] R[100]mm/sec CNT100;
   1:  PR[91,1] = PR[90,1] + 22.751;
   1:  PR[91,2] = PR[90,2] + -28.821;
   1:  PR[91,3] = PR[90,3] + 133.023;
   1:L PR[91] R[100]mm/sec CNT100;
   1:  PR[91,1] = PR[90,1] + 25.029;
   1:  PR[91,2] = PR[90,2] + -29.861;
   1:  PR[91,3] = PR[90,3] + 133.031;
   1:L PR[91] R[100]mm/sec CNT100;
   1:  PR[91,1] = PR[90,1] + 27.403;
   1:  PR[91,2] = PR[90,2] + -30.837;
   1:  PR[91,3] = PR[90,3] + 133.046;
   1:L PR[91] R[100]mm/sec CNT100;
   1:  PR[91,1] = PR[90,1] + 31.252;
   1:  PR[91,2] = PR[90,2] + -32.112;
   1:  PR[91,3] = PR[90,3] + 133.060;
   1:L PR[91] R[100]mm/sec CNT100;
   1:  PR[91,1] = PR[90,1] + 32.283;
   1:  PR[91,2] = PR[90,2] + -32.348;
   1:  PR[91,3] = PR[90,3] + 133.083;
   1:L PR[91] R[100]mm/sec CNT100;
   1:  PR[91,1] = PR[90,1] + 35.894;
   1:  PR[91,2] = PR[90,2] + -33.096;
   1:  PR[91,3] = PR[90,3] + 133.089;
   1:L PR[91] R[100]mm/sec CNT100;
   1:  PR[91,1] = PR[90,1] + 36.448;
   1:  PR[91,2] = PR[90,2] + -33.198;
   1:  PR[91,3] = PR[90,3] + 133.110;
   1:L PR[91] R[100]mm/sec CNT100;
   1:  PR[91,1] = PR[90,1] + 40.619;
   1:  PR[91,2] = PR[90,2] + -33.612;
   1:  PR[91,3] = PR[90,3] + 133.113;
   1:L PR[91] R[100]mm/sec CNT100;
   1:  PR[91,1] = PR[90,1] + 41.865;
   1:  PR[91,2] = PR[90,2] + -33.688;
   1:  PR[91,3] = PR[90,3] + 133.136;
   1:L PR[91] R[100]mm/sec CNT100;
   1:  PR[91,1] = PR[90,1] + 45.866;
   1:  PR[91,2] = PR[90,2] + -33.652;
   1:  PR[91,3] = PR[90,3] + 133.143;
   1:L PR[91] R[100]mm/sec CNT100;
   1:  PR[91,1] = PR[90,1] + 47.670;
   1:  PR[91,2] = PR[90,2] + -33.542;
   1:  PR[91,3] = PR[90,3] + 133.166;
   1:L PR[91] R[100]mm/sec CNT100;
   1:  PR[91,1] = PR[90,1] + 51.223;
   1:  PR[91,2] = PR[90,2] + -33.109;
   1:  PR[91,3] = PR[90,3] + 133.176;
   1:L PR[91] R[100]mm/sec CNT100;
   1:  PR[91,1] = PR[90,1] + 53.393;
   1:  PR[91,2] = PR[90,2] + -32.708;
   1:  PR[91,3] = PR[90,3] + 133.196;
   1:L PR[91] R[100]mm/sec CNT100;
   1:  PR[91,1] = PR[90,1] + 56.474;
   1:  PR[91,2] = PR[90,2] + -31.970;
   1:  PR[91,3] = PR[90,3] + 133.209;
   1:L PR[91] R[100]mm/sec CNT100;
   1:  PR[91,1] = PR[90,1] + 58.944;
   1:  PR[91,2] = PR[90,2] + -31.051;
   1:  PR[91,3] = PR[90,3] + 133.227;
   1:L PR[91] R[100]mm/sec CNT100;
   1:  PR[91,1] = PR[90,1] + 64.062;
   1:  PR[91,2] = PR[90,2] + -29.091;
   1:  PR[91,3] = PR[90,3] + 133.241;
   1:L PR[91] R[100]mm/sec CNT100;
   1:  PR[91,1] = PR[90,1] + 66.308;
   1:  PR[91,2] = PR[90,2] + -27.943;
   1:  PR[91,3] = PR[90,3] + 133.272;
   1:L PR[91] R[100]mm/sec CNT100;
   1:  PR[91,1] = PR[90,1] + 68.137;
   1:  PR[91,2] = PR[90,2] + -26.687;
   1:  PR[91,3] = PR[90,3] + 133.287;
   1:L PR[91] R[100]mm/sec CNT100;
   1:  PR[91,1] = PR[90,1] + 72.735;
   1:  PR[91,2] = PR[90,2] + -23.419;
   1:  PR[91,3] = PR[90,3] + 133.299;
   1:L PR[91] R[100]mm/sec CNT100;
   1:  PR[91,1] = PR[90,1] + 74.267;
   1:  PR[91,2] = PR[90,2] + -22.045;
   1:  PR[91,3] = PR[90,3] + 133.331;
   1:L PR[91] R[100]mm/sec CNT100;
   1:  PR[91,1] = PR[90,1] + 75.497;
   1:  PR[91,2] = PR[90,2] + -20.581;
   1:  PR[91,3] = PR[90,3] + 133.342;
   1:L PR[91] R[100]mm/sec CNT100;
   1:  PR[91,1] = PR[90,1] + 78.953;
   1:  PR[91,2] = PR[90,2] + -16.407;
   1:  PR[91,3] = PR[90,3] + 133.353;
   1:L PR[91] R[100]mm/sec CNT100;
   1:  PR[91,1] = PR[90,1] + 79.858;
   1:  PR[91,2] = PR[90,2] + -14.946;
   1:  PR[91,3] = PR[90,3] + 133.384;
   1:L PR[91] R[100]mm/sec CNT100;
   1:  PR[91,1] = PR[90,1] + 80.535;
   1:  PR[91,2] = PR[90,2] + -13.346;
   1:  PR[91,3] = PR[90,3] + 133.393;
   1:L PR[91] R[100]mm/sec CNT100;
   1:  PR[91,1] = PR[90,1] + 82.619;
   1:  PR[91,2] = PR[90,2] + -8.682;
   1:  PR[91,3] = PR[90,3] + 133.403;
   1:L PR[91] R[100]mm/sec CNT100;
   1:  PR[91,1] = PR[90,1] + 82.983;
   1:  PR[91,2] = PR[90,2] + -7.218;
   1:  PR[91,3] = PR[90,3] + 133.432;
   1:L PR[91] R[100]mm/sec CNT100;
   1:  PR[91,1] = PR[90,1] + 83.121;
   1:  PR[91,2] = PR[90,2] + -5.515;
   1:  PR[91,3] = PR[90,3] + 133.441;
   1:L PR[91] R[100]mm/sec CNT100;
   1:  PR[91,1] = PR[90,1] + 83.808;
   1:  PR[91,2] = PR[90,2] + -0.670;
   1:  PR[91,3] = PR[90,3] + 133.450;
   1:L PR[91] R[100]mm/sec CNT100;
   1:  PR[91,1] = PR[90,1] + 83.682;
   1:  PR[91,2] = PR[90,2] + 0.868;
   1:  PR[91,3] = PR[90,3] + 133.478;
   1:L PR[91] R[100]mm/sec CNT100;
   1:  PR[91,1] = PR[90,1] + 82.997;
   1:  PR[91,2] = PR[90,2] + 5.702;
   1:  PR[91,3] = PR[90,3] + 133.486;
   1:L PR[91] R[100]mm/sec CNT100;
   1:  PR[91,1] = PR[90,1] + 82.614;
   1:  PR[91,2] = PR[90,2] + 7.242;
   1:  PR[91,3] = PR[90,3] + 133.514;
   1:L PR[91] R[100]mm/sec CNT100;
   1:  PR[91,1] = PR[90,1] + 81.922;
   1:  PR[91,2] = PR[90,2] + 8.873;
   1:  PR[91,3] = PR[90,3] + 133.523;
   1:L PR[91] R[100]mm/sec CNT100;
   1:  PR[91,1] = PR[90,1] + 79.868;
   1:  PR[91,2] = PR[90,2] + 13.472;
   1:  PR[91,3] = PR[90,3] + 133.533;
   1:L PR[91] R[100]mm/sec CNT100;
   1:  PR[91,1] = PR[90,1] + 78.953;
   1:  PR[91,2] = PR[90,2] + 14.948;
   1:  PR[91,3] = PR[90,3] + 133.561;
   1:L PR[91] R[100]mm/sec CNT100;
   1:  PR[91,1] = PR[90,1] + 74.262;
   1:  PR[91,2] = PR[90,2] + 20.591;
   1:  PR[91,3] = PR[90,3] + 133.571;
   1:L PR[91] R[100]mm/sec CNT100;
   1:  PR[91,1] = PR[90,1] + 72.744;
   1:  PR[91,2] = PR[90,2] + 21.952;
   1:  PR[91,3] = PR[90,3] + 133.612;
   1:L PR[91] R[100]mm/sec CNT100;
   1:  PR[91,1] = PR[90,1] + 70.645;
   1:  PR[91,2] = PR[90,2] + 23.400;
   1:  PR[91,3] = PR[90,3] + 133.624;
   1:L PR[91] R[100]mm/sec CNT100;
   1:  PR[91,1] = PR[90,1] + 66.292;
   1:  PR[91,2] = PR[90,2] + 26.492;
   1:  PR[91,3] = PR[90,3] + 133.638;
   1:L PR[91] R[100]mm/sec CNT100;
   1:  PR[91,1] = PR[90,1] + 64.068;
   1:  PR[91,2] = PR[90,2] + 27.630;
   1:  PR[91,3] = PR[90,3] + 133.668;
   1:L PR[91] R[100]mm/sec CNT100;
   1:  PR[91,1] = PR[90,1] + 61.088;
   1:  PR[91,2] = PR[90,2] + 28.744;
   1:  PR[91,3] = PR[90,3] + 133.682;
   1:L PR[91] R[100]mm/sec CNT100;
   1:  PR[91,1] = PR[90,1] + 56.463;
   1:  PR[91,2] = PR[90,2] + 30.514;
   1:  PR[91,3] = PR[90,3] + 133.700;
   1:L PR[91] R[100]mm/sec CNT100;
   1:  PR[91,1] = PR[90,1] + 53.391;
   1:  PR[91,2] = PR[90,2] + 31.250;
   1:  PR[91,3] = PR[90,3] + 133.728;
   1:L PR[91] R[100]mm/sec CNT100;
   1:  PR[91,1] = PR[90,1] + 51.221;
   1:  PR[91,2] = PR[90,2] + 31.650;
   1:  PR[91,3] = PR[90,3] + 133.746;
   1:L PR[91] R[100]mm/sec CNT100;
   1:  PR[91,1] = PR[90,1] + 47.668;
   1:  PR[91,2] = PR[90,2] + 32.083;
   1:  PR[91,3] = PR[90,3] + 133.758;
   1:L PR[91] R[100]mm/sec CNT100;
   1:  PR[91,1] = PR[90,1] + 45.864;
   1:  PR[91,2] = PR[90,2] + 32.193;
   1:  PR[91,3] = PR[90,3] + 133.779;
   1:L PR[91] R[100]mm/sec CNT100;
   1:  PR[91,1] = PR[90,1] + 41.864;
   1:  PR[91,2] = PR[90,2] + 32.230;
   1:  PR[91,3] = PR[90,3] + 133.789;
   1:L PR[91] R[100]mm/sec CNT100;
   1:  PR[91,1] = PR[90,1] + 40.617;
   1:  PR[91,2] = PR[90,2] + 32.153;
   1:  PR[91,3] = PR[90,3] + 133.811;
   1:L PR[91] R[100]mm/sec CNT100;
   1:  PR[91,1] = PR[90,1] + 36.447;
   1:  PR[91,2] = PR[90,2] + 31.739;
   1:  PR[91,3] = PR[90,3] + 133.818;
   1:L PR[91] R[100]mm/sec CNT100;
   1:  PR[91,1] = PR[90,1] + 35.894;
   1:  PR[91,2] = PR[90,2] + 31.637;
   1:  PR[91,3] = PR[90,3] + 133.842;
   1:L PR[91] R[100]mm/sec CNT100;
   1:  PR[91,1] = PR[90,1] + 32.283;
   1:  PR[91,2] = PR[90,2] + 30.889;
   1:  PR[91,3] = PR[90,3] + 133.845;
   1:L PR[91] R[100]mm/sec CNT100;
   1:  PR[91,1] = PR[90,1] + 31.253;
   1:  PR[91,2] = PR[90,2] + 30.653;
   1:  PR[91,3] = PR[90,3] + 133.866;
   1:L PR[91] R[100]mm/sec CNT100;
   1:  PR[91,1] = PR[90,1] + 27.405;
   1:  PR[91,2] = PR[90,2] + 29.378;
   1:  PR[91,3] = PR[90,3] + 133.872;
   1:L PR[91] R[100]mm/sec CNT100;
   1:  PR[91,1] = PR[90,1] + 25.032;
   1:  PR[91,2] = PR[90,2] + 28.404;
   1:  PR[91,3] = PR[90,3] + 133.895;
   1:L PR[91] R[100]mm/sec CNT100;
   1:  PR[91,1] = PR[90,1] + 22.748;
   1:  PR[91,2] = PR[90,2] + 27.361;
   1:  PR[91,3] = PR[90,3] + 133.909;
   1:L PR[91] R[100]mm/sec CNT100;
   1:  PR[91,1] = PR[90,1] + 17.409;
   1:  PR[91,2] = PR[90,2] + 24.148;
   1:  PR[91,3] = PR[90,3] + 133.923;
   1:L PR[91] R[100]mm/sec CNT100;
   1:  PR[91,1] = PR[90,1] + 12.724;
   1:  PR[91,2] = PR[90,2] + 20.320;
   1:  PR[91,3] = PR[90,3] + 133.958;
   1:L PR[91] R[100]mm/sec CNT100;
   1:  PR[91,1] = PR[90,1] + 10.218;
   1:  PR[91,2] = PR[90,2] + 17.553;
   1:  PR[91,3] = PR[90,3] + 133.993;
   1:L PR[91] R[100]mm/sec CNT100;
   1:  PR[91,1] = PR[90,1] + 8.746;
   1:  PR[91,2] = PR[90,2] + 15.849;
   1:  PR[91,3] = PR[90,3] + 134.014;
   1:L PR[91] R[100]mm/sec CNT100;
   1:  PR[91,1] = PR[90,1] + 6.134;
   1:  PR[91,2] = PR[90,2] + 11.517;
   1:  PR[91,3] = PR[90,3] + 134.026;
   1:L PR[91] R[100]mm/sec CNT100;
   1:  PR[91,1] = PR[90,1] + 5.522;
   1:  PR[91,2] = PR[90,2] + 10.610;
   1:  PR[91,3] = PR[90,3] + 134.055;
   1:L PR[91] R[100]mm/sec CNT100;
   1:  PR[91,1] = PR[90,1] + 3.342;
   1:  PR[91,2] = PR[90,2] + 4.978;
   1:  PR[91,3] = PR[90,3] + 134.061;
   1:L PR[91] R[100]mm/sec CNT100;
   1:  PR[91] = PR[90];
   1:  PR[91,1] = PR[90,1] + 3.828;
   1:  PR[91,2] = PR[90,2] + -0.729;
   1:  PR[91,3] = PR[90,3] + 135.395;
   1:L PR[91] R[100]mm/sec CNT100;
   1:  PR[91,1] = PR[90,1] + 4.535;
   1:  PR[91,2] = PR[90,2] + -6.481;
   1:  PR[91,3] = PR[90,3] + 134.128;
   1:L PR[91] R[100]mm/sec CNT100;
   1:  PR[91,1] = PR[90,1] + 5.187;
   1:  PR[91,2] = PR[90,2] + -8.163;
   1:  PR[91,3] = PR[90,3] + 134.160;
   1:L PR[91] R[100]mm/sec CNT100;
   1:  PR[91,1] = PR[90,1] + 6.557;
   1:  PR[91,2] = PR[90,2] + -12.126;
   1:  PR[91,3] = PR[90,3] + 134.171;
   1:L PR[91] R[100]mm/sec CNT100;
   1:  PR[91,1] = PR[90,1] + 7.054;
   1:  PR[91,2] = PR[90,2] + -12.989;
   1:  PR[91,3] = PR[90,3] + 134.194;
   1:L PR[91] R[100]mm/sec CNT100;
   1:  PR[91,1] = PR[90,1] + 9.589;
   1:  PR[91,2] = PR[90,2] + -17.194;
   1:  PR[91,3] = PR[90,3] + 134.200;
   1:L PR[91] R[100]mm/sec CNT100;
   1:  PR[91,1] = PR[90,1] + 12.246;
   1:  PR[91,2] = PR[90,2] + -20.272;
   1:  PR[91,3] = PR[90,3] + 134.228;
   1:L PR[91] R[100]mm/sec CNT100;
   1:  PR[91,1] = PR[90,1] + 13.511;
   1:  PR[91,2] = PR[90,2] + -21.668;
   1:  PR[91,3] = PR[90,3] + 134.250;
   1:L PR[91] R[100]mm/sec CNT100;
   1:  PR[91,1] = PR[90,1] + 15.933;
   1:  PR[91,2] = PR[90,2] + -23.645;
   1:  PR[91,3] = PR[90,3] + 134.261;
   1:L PR[91] R[100]mm/sec CNT100;
   1:  PR[91,1] = PR[90,1] + 17.904;
   1:  PR[91,2] = PR[90,2] + -25.332;
   1:  PR[91,3] = PR[90,3] + 134.279;
   1:L PR[91] R[100]mm/sec CNT100;
   1:  PR[91,1] = PR[90,1] + 18.407;
   1:  PR[91,2] = PR[90,2] + -25.723;
   1:  PR[91,3] = PR[90,3] + 134.293;
   1:L PR[91] R[100]mm/sec CNT100;
   1:  PR[91,1] = PR[90,1] + 21.712;
   1:  PR[91,2] = PR[90,2] + -27.696;
   1:  PR[91,3] = PR[90,3] + 134.297;
   1:L PR[91] R[100]mm/sec CNT100;
   1:  PR[91,1] = PR[90,1] + 23.469;
   1:  PR[91,2] = PR[90,2] + -28.771;
   1:  PR[91,3] = PR[90,3] + 134.319;
   1:L PR[91] R[100]mm/sec CNT100;
   1:  PR[91,1] = PR[90,1] + 26.681;
   1:  PR[91,2] = PR[90,2] + -30.237;
   1:  PR[91,3] = PR[90,3] + 134.330;
   1:L PR[91] R[100]mm/sec CNT100;
   1:  PR[91,1] = PR[90,1] + 27.893;
   1:  PR[91,2] = PR[90,2] + -30.736;
   1:  PR[91,3] = PR[90,3] + 134.350;
   1:L PR[91] R[100]mm/sec CNT100;
   1:  PR[91,1] = PR[90,1] + 30.523;
   1:  PR[91,2] = PR[90,2] + -31.607;
   1:  PR[91,3] = PR[90,3] + 134.358;
   1:L PR[91] R[100]mm/sec CNT100;
   1:  PR[91,1] = PR[90,1] + 31.797;
   1:  PR[91,2] = PR[90,2] + -31.976;
   1:  PR[91,3] = PR[90,3] + 134.373;
   1:L PR[91] R[100]mm/sec CNT100;
   1:  PR[91,1] = PR[90,1] + 32.318;
   1:  PR[91,2] = PR[90,2] + -32.176;
   1:  PR[91,3] = PR[90,3] + 134.381;
   1:L PR[91] R[100]mm/sec CNT100;
   1:  PR[91,1] = PR[90,1] + 36.433;
   1:  PR[91,2] = PR[90,2] + -33.028;
   1:  PR[91,3] = PR[90,3] + 134.384;
   1:L PR[91] R[100]mm/sec CNT100;
   1:  PR[91,1] = PR[90,1] + 37.431;
   1:  PR[91,2] = PR[90,2] + -33.212;
   1:  PR[91,3] = PR[90,3] + 134.408;
   1:L PR[91] R[100]mm/sec CNT100;
   1:  PR[91,1] = PR[90,1] + 41.243;
   1:  PR[91,2] = PR[90,2] + -33.591;
   1:  PR[91,3] = PR[90,3] + 134.413;
   1:L PR[91] R[100]mm/sec CNT100;
   1:  PR[91,1] = PR[90,1] + 42.892;
   1:  PR[91,2] = PR[90,2] + -33.692;
   1:  PR[91,3] = PR[90,3] + 134.435;
   1:L PR[91] R[100]mm/sec CNT100;
   1:  PR[91,1] = PR[90,1] + 46.548;
   1:  PR[91,2] = PR[90,2] + -33.659;
   1:  PR[91,3] = PR[90,3] + 134.444;
   1:L PR[91] R[100]mm/sec CNT100;
   1:  PR[91,1] = PR[90,1] + 48.707;
   1:  PR[91,2] = PR[90,2] + -33.526;
   1:  PR[91,3] = PR[90,3] + 134.465;
   1:L PR[91] R[100]mm/sec CNT100;
   1:  PR[91,1] = PR[90,1] + 51.953;
   1:  PR[91,2] = PR[90,2] + -33.131;
   1:  PR[91,3] = PR[90,3] + 134.477;
   1:L PR[91] R[100]mm/sec CNT100;
   1:  PR[91,1] = PR[90,1] + 54.431;
   1:  PR[91,2] = PR[90,2] + -32.674;
   1:  PR[91,3] = PR[90,3] + 134.496;
   1:L PR[91] R[100]mm/sec CNT100;
   1:  PR[91,1] = PR[90,1] + 57.241;
   1:  PR[91,2] = PR[90,2] + -32.001;
   1:  PR[91,3] = PR[90,3] + 134.510;
   1:L PR[91] R[100]mm/sec CNT100;
   1:  PR[91,1] = PR[90,1] + 59.494;
   1:  PR[91,2] = PR[90,2] + -31.162;
   1:  PR[91,3] = PR[90,3] + 134.526;
   1:L PR[91] R[100]mm/sec CNT100;
   1:  PR[91,1] = PR[90,1] + 65.078;
   1:  PR[91,2] = PR[90,2] + -29.024;
   1:  PR[91,3] = PR[90,3] + 134.540;
   1:L PR[91] R[100]mm/sec CNT100;
   1:  PR[91,1] = PR[90,1] + 67.118;
   1:  PR[91,2] = PR[90,2] + -27.980;
   1:  PR[91,3] = PR[90,3] + 134.573;
   1:L PR[91] R[100]mm/sec CNT100;
   1:  PR[91,1] = PR[90,1] + 68.785;
   1:  PR[91,2] = PR[90,2] + -26.836;
   1:  PR[91,3] = PR[90,3] + 134.586;
   1:L PR[91] R[100]mm/sec CNT100;
   1:  PR[91,1] = PR[90,1] + 73.706;
   1:  PR[91,2] = PR[90,2] + -23.339;
   1:  PR[91,3] = PR[90,3] + 134.598;
   1:L PR[91] R[100]mm/sec CNT100;
   1:  PR[91,1] = PR[90,1] + 75.091;
   1:  PR[91,2] = PR[90,2] + -22.097;
   1:  PR[91,3] = PR[90,3] + 134.632;
   1:L PR[91] R[100]mm/sec CNT100;
   1:  PR[91,1] = PR[90,1] + 79.878;
   1:  PR[91,2] = PR[90,2] + -16.336;
   1:  PR[91,3] = PR[90,3] + 134.642;
   1:L PR[91] R[100]mm/sec CNT100;
   1:  PR[91,1] = PR[90,1] + 80.694;
   1:  PR[91,2] = PR[90,2] + -15.019;
   1:  PR[91,3] = PR[90,3] + 134.684;
   1:L PR[91] R[100]mm/sec CNT100;
   1:  PR[91,1] = PR[90,1] + 81.310;
   1:  PR[91,2] = PR[90,2] + -13.562;
   1:  PR[91,3] = PR[90,3] + 134.693;
   1:L PR[91] R[100]mm/sec CNT100;
   1:  PR[91,1] = PR[90,1] + 83.508;
   1:  PR[91,2] = PR[90,2] + -8.641;
   1:  PR[91,3] = PR[90,3] + 134.702;
   1:L PR[91] R[100]mm/sec CNT100;
   1:  PR[91,1] = PR[90,1] + 83.835;
   1:  PR[91,2] = PR[90,2] + -7.327;
   1:  PR[91,3] = PR[90,3] + 134.733;
   1:L PR[91] R[100]mm/sec CNT100;
   1:  PR[91,1] = PR[90,1] + 83.961;
   1:  PR[91,2] = PR[90,2] + -5.776;
   1:  PR[91,3] = PR[90,3] + 134.740;
   1:L PR[91] R[100]mm/sec CNT100;
   1:  PR[91,1] = PR[90,1] + 84.685;
   1:  PR[91,2] = PR[90,2] + -0.670;
   1:  PR[91,3] = PR[90,3] + 134.749;
   1:L PR[91] R[100]mm/sec CNT100;
   1:  PR[91,1] = PR[90,1] + 84.572;
   1:  PR[91,2] = PR[90,2] + 0.716;
   1:  PR[91,3] = PR[90,3] + 134.778;
   1:L PR[91] R[100]mm/sec CNT100;
   1:  PR[91,1] = PR[90,1] + 83.849;
   1:  PR[91,2] = PR[90,2] + 5.811;
   1:  PR[91,3] = PR[90,3] + 134.786;
   1:L PR[91] R[100]mm/sec CNT100;
   1:  PR[91,1] = PR[90,1] + 83.503;
   1:  PR[91,2] = PR[90,2] + 7.201;
   1:  PR[91,3] = PR[90,3] + 134.815;
   1:L PR[91] R[100]mm/sec CNT100;
   1:  PR[91,1] = PR[90,1] + 82.875;
   1:  PR[91,2] = PR[90,2] + 8.682;
   1:  PR[91,3] = PR[90,3] + 134.823;
   1:L PR[91] R[100]mm/sec CNT100;
   1:  PR[91,1] = PR[90,1] + 80.703;
   1:  PR[91,2] = PR[90,2] + 13.544;
   1:  PR[91,3] = PR[90,3] + 134.832;
   1:L PR[91] R[100]mm/sec CNT100;
   1:  PR[91,1] = PR[90,1] + 79.877;
   1:  PR[91,2] = PR[90,2] + 14.878;
   1:  PR[91,3] = PR[90,3] + 134.862;
   1:L PR[91] R[100]mm/sec CNT100;
   1:  PR[91,1] = PR[90,1] + 75.089;
   1:  PR[91,2] = PR[90,2] + 20.640;
   1:  PR[91,3] = PR[90,3] + 134.871;
   1:L PR[91] R[100]mm/sec CNT100;
   1:  PR[91,1] = PR[90,1] + 73.715;
   1:  PR[91,2] = PR[90,2] + 21.872;
   1:  PR[91,3] = PR[90,3] + 134.913;
   1:L PR[91] R[100]mm/sec CNT100;
   1:  PR[91,1] = PR[90,1] + 71.799;
   1:  PR[91,2] = PR[90,2] + 23.193;
   1:  PR[91,3] = PR[90,3] + 134.924;
   1:L PR[91] R[100]mm/sec CNT100;
   1:  PR[91,1] = PR[90,1] + 67.102;
   1:  PR[91,2] = PR[90,2] + 26.530;
   1:  PR[91,3] = PR[90,3] + 134.937;
   1:L PR[91] R[100]mm/sec CNT100;
   1:  PR[91,1] = PR[90,1] + 65.083;
   1:  PR[91,2] = PR[90,2] + 27.562;
   1:  PR[91,3] = PR[90,3] + 134.969;
   1:L PR[91] R[100]mm/sec CNT100;
   1:  PR[91,1] = PR[90,1] + 62.361;
   1:  PR[91,2] = PR[90,2] + 28.580;
   1:  PR[91,3] = PR[90,3] + 134.982;
   1:L PR[91] R[100]mm/sec CNT100;
   1:  PR[91,1] = PR[90,1] + 57.230;
   1:  PR[91,2] = PR[90,2] + 30.545;
   1:  PR[91,3] = PR[90,3] + 134.998;
   1:L PR[91] R[100]mm/sec CNT100;
   1:  PR[91,1] = PR[90,1] + 54.428;
   1:  PR[91,2] = PR[90,2] + 31.215;
   1:  PR[91,3] = PR[90,3] + 135.029;
   1:L PR[91] R[100]mm/sec CNT100;
   1:  PR[91,1] = PR[90,1] + 51.951;
   1:  PR[91,2] = PR[90,2] + 31.672;
   1:  PR[91,3] = PR[90,3] + 135.046;
   1:L PR[91] R[100]mm/sec CNT100;
   1:  PR[91,1] = PR[90,1] + 48.705;
   1:  PR[91,2] = PR[90,2] + 32.068;
   1:  PR[91,3] = PR[90,3] + 135.060;
   1:L PR[91] R[100]mm/sec CNT100;
   1:  PR[91,1] = PR[90,1] + 46.546;
   1:  PR[91,2] = PR[90,2] + 32.200;
   1:  PR[91,3] = PR[90,3] + 135.078;
   1:L PR[91] R[100]mm/sec CNT100;
   1:  PR[91,1] = PR[90,1] + 42.890;
   1:  PR[91,2] = PR[90,2] + 32.233;
   1:  PR[91,3] = PR[90,3] + 135.091;
   1:L PR[91] R[100]mm/sec CNT100;
   1:  PR[91,1] = PR[90,1] + 41.241;
   1:  PR[91,2] = PR[90,2] + 32.132;
   1:  PR[91,3] = PR[90,3] + 135.111;
   1:L PR[91] R[100]mm/sec CNT100;
   1:  PR[91,1] = PR[90,1] + 37.430;
   1:  PR[91,2] = PR[90,2] + 31.754;
   1:  PR[91,3] = PR[90,3] + 135.120;
   1:L PR[91] R[100]mm/sec CNT100;
   1:  PR[91,1] = PR[90,1] + 36.433;
   1:  PR[91,2] = PR[90,2] + 31.569;
   1:  PR[91,3] = PR[90,3] + 135.142;
   1:L PR[91] R[100]mm/sec CNT100;
   1:  PR[91,1] = PR[90,1] + 32.263;
   1:  PR[91,2] = PR[90,2] + 30.705;
   1:  PR[91,3] = PR[90,3] + 135.148;
   1:L PR[91] R[100]mm/sec CNT100;
   1:  PR[91,1] = PR[90,1] + 30.549;
   1:  PR[91,2] = PR[90,2] + 30.157;
   1:  PR[91,3] = PR[90,3] + 135.172;
   1:L PR[91] R[100]mm/sec CNT100;
   1:  PR[91,1] = PR[90,1] + 27.894;
   1:  PR[91,2] = PR[90,2] + 29.277;
   1:  PR[91,3] = PR[90,3] + 135.182;
   1:L PR[91] R[100]mm/sec CNT100;
   1:  PR[91,1] = PR[90,1] + 26.683;
   1:  PR[91,2] = PR[90,2] + 28.780;
   1:  PR[91,3] = PR[90,3] + 135.198;
   1:L PR[91] R[100]mm/sec CNT100;
   1:  PR[91,1] = PR[90,1] + 23.466;
   1:  PR[91,2] = PR[90,2] + 27.311;
   1:  PR[91,3] = PR[90,3] + 135.205;
   1:L PR[91] R[100]mm/sec CNT100;
   1:  PR[91,1] = PR[90,1] + 18.414;
   1:  PR[91,2] = PR[90,2] + 24.269;
   1:  PR[91,3] = PR[90,3] + 135.225;
   1:L PR[91] R[100]mm/sec CNT100;
   1:  PR[91,1] = PR[90,1] + 17.907;
   1:  PR[91,2] = PR[90,2] + 23.875;
   1:  PR[91,3] = PR[90,3] + 135.258;
   1:L PR[91] R[100]mm/sec CNT100;
   1:  PR[91,1] = PR[90,1] + 15.933;
   1:  PR[91,2] = PR[90,2] + 22.186;
   1:  PR[91,3] = PR[90,3] + 135.262;
   1:L PR[91] R[100]mm/sec CNT100;
   1:  PR[91,1] = PR[90,1] + 13.514;
   1:  PR[91,2] = PR[90,2] + 20.213;
   1:  PR[91,3] = PR[90,3] + 135.277;
   1:L PR[91] R[100]mm/sec CNT100;
   1:  PR[91,1] = PR[90,1] + 12.251;
   1:  PR[91,2] = PR[90,2] + 18.818;
   1:  PR[91,3] = PR[90,3] + 135.294;
   1:L PR[91] R[100]mm/sec CNT100;
   1:  PR[91,1] = PR[90,1] + 9.592;
   1:  PR[91,2] = PR[90,2] + 15.739;
   1:  PR[91,3] = PR[90,3] + 135.305;
   1:L PR[91] R[100]mm/sec CNT100;
   1:  PR[91,1] = PR[90,1] + 7.057;
   1:  PR[91,2] = PR[90,2] + 11.535;
   1:  PR[91,3] = PR[90,3] + 135.328;
   1:L PR[91] R[100]mm/sec CNT100;
   1:  PR[91,1] = PR[90,1] + 6.558;
   1:  PR[91,2] = PR[90,2] + 10.671;
   1:  PR[91,3] = PR[90,3] + 135.356;
   1:L PR[91] R[100]mm/sec CNT100;
   1:  PR[91,1] = PR[90,1] + 5.187;
   1:  PR[91,2] = PR[90,2] + 6.704;
   1:  PR[91,3] = PR[90,3] + 135.361;
   1:L PR[91] R[100]mm/sec CNT100;
   1:  PR[91,1] = PR[90,1] + 4.536;
   1:  PR[91,2] = PR[90,2] + 5.024;
   1:  PR[91,3] = PR[90,3] + 135.385;
   1:L PR[91] R[100]mm/sec CNT100;
   1:  PR[91] = PR[90];
   1:  PR[91,1] = PR[90,1] + 4.940;
   1:  PR[91,2] = PR[90,2] + -0.289;
   1:  PR[91,3] = PR[90,3] + 136.695;
   1:L PR[91] R[100]mm/sec CNT100;
   1:  PR[91,1] = PR[90,1] + 4.910;
   1:  PR[91,2] = PR[90,2] + -0.687;
   1:  PR[91,3] = PR[90,3] + 135.425;
   1:L PR[91] R[100]mm/sec CNT100;
   1:  PR[91,1] = PR[90,1] + 5.401;
   1:  PR[91,2] = PR[90,2] + -4.870;
   1:  PR[91,3] = PR[90,3] + 135.428;
   1:L PR[91] R[100]mm/sec CNT100;
   1:  PR[91,1] = PR[90,1] + 5.563;
   1:  PR[91,2] = PR[90,2] + -6.534;
   1:  PR[91,3] = PR[90,3] + 135.451;
   1:L PR[91] R[100]mm/sec CNT100;
   1:  PR[91,1] = PR[90,1] + 5.829;
   1:  PR[91,2] = PR[90,2] + -7.339;
   1:  PR[91,3] = PR[90,3] + 135.461;
   1:L PR[91] R[100]mm/sec CNT100;
   1:  PR[91,1] = PR[90,1] + 7.453;
   1:  PR[91,2] = PR[90,2] + -12.037;
   1:  PR[91,3] = PR[90,3] + 135.466;
   1:L PR[91] R[100]mm/sec CNT100;
   1:  PR[91,1] = PR[90,1] + 8.815;
   1:  PR[91,2] = PR[90,2] + -14.397;
   1:  PR[91,3] = PR[90,3] + 135.494;
   1:L PR[91] R[100]mm/sec CNT100;
   1:  PR[91,1] = PR[90,1] + 10.435;
   1:  PR[91,2] = PR[90,2] + -17.085;
   1:  PR[91,3] = PR[90,3] + 135.509;
   1:L PR[91] R[100]mm/sec CNT100;
   1:  PR[91,1] = PR[90,1] + 14.334;
   1:  PR[91,2] = PR[90,2] + -21.593;
   1:  PR[91,3] = PR[90,3] + 135.527;
   1:L PR[91] R[100]mm/sec CNT100;
   1:  PR[91,1] = PR[90,1] + 18.292;
   1:  PR[91,2] = PR[90,2] + -24.969;
   1:  PR[91,3] = PR[90,3] + 135.560;
   1:L PR[91] R[100]mm/sec CNT100;
   1:  PR[91,1] = PR[90,1] + 19.392;
   1:  PR[91,2] = PR[90,2] + -25.825;
   1:  PR[91,3] = PR[90,3] + 135.590;
   1:L PR[91] R[100]mm/sec CNT100;
   1:  PR[91,1] = PR[90,1] + 21.915;
   1:  PR[91,2] = PR[90,2] + -27.331;
   1:  PR[91,3] = PR[90,3] + 135.598;
   1:L PR[91] R[100]mm/sec CNT100;
   1:  PR[91,1] = PR[90,1] + 24.187;
   1:  PR[91,2] = PR[90,2] + -28.720;
   1:  PR[91,3] = PR[90,3] + 135.614;
   1:L PR[91] R[100]mm/sec CNT100;
   1:  PR[91,1] = PR[90,1] + 28.290;
   1:  PR[91,2] = PR[90,2] + -30.594;
   1:  PR[91,3] = PR[90,3] + 135.629;
   1:L PR[91] R[100]mm/sec CNT100;
   1:  PR[91,1] = PR[90,1] + 28.618;
   1:  PR[91,2] = PR[90,2] + -30.711;
   1:  PR[91,3] = PR[90,3] + 135.655;
   1:L PR[91] R[100]mm/sec CNT100;
   1:  PR[91,1] = PR[90,1] + 31.797;
   1:  PR[91,2] = PR[90,2] + -31.633;
   1:  PR[91,3] = PR[90,3] + 135.657;
   1:L PR[91] R[100]mm/sec CNT100;
   1:  PR[91,1] = PR[90,1] + 33.249;
   1:  PR[91,2] = PR[90,2] + -32.189;
   1:  PR[91,3] = PR[90,3] + 135.675;
   1:L PR[91] R[100]mm/sec CNT100;
   1:  PR[91,1] = PR[90,1] + 36.973;
   1:  PR[91,2] = PR[90,2] + -32.961;
   1:  PR[91,3] = PR[90,3] + 135.684;
   1:L PR[91] R[100]mm/sec CNT100;
   1:  PR[91,1] = PR[90,1] + 38.415;
   1:  PR[91,2] = PR[90,2] + -33.227;
   1:  PR[91,3] = PR[90,3] + 135.706;
   1:L PR[91] R[100]mm/sec CNT100;
   1:  PR[91,1] = PR[90,1] + 41.868;
   1:  PR[91,2] = PR[90,2] + -33.570;
   1:  PR[91,3] = PR[90,3] + 135.714;
   1:L PR[91] R[100]mm/sec CNT100;
   1:  PR[91,1] = PR[90,1] + 43.918;
   1:  PR[91,2] = PR[90,2] + -33.695;
   1:  PR[91,3] = PR[90,3] + 135.734;
   1:L PR[91] R[100]mm/sec CNT100;
   1:  PR[91,1] = PR[90,1] + 47.230;
   1:  PR[91,2] = PR[90,2] + -33.665;
   1:  PR[91,3] = PR[90,3] + 135.745;
   1:L PR[91] R[100]mm/sec CNT100;
   1:  PR[91,1] = PR[90,1] + 49.744;
   1:  PR[91,2] = PR[90,2] + -33.511;
   1:  PR[91,3] = PR[90,3] + 135.764;
   1:L PR[91] R[100]mm/sec CNT100;
   1:  PR[91,1] = PR[90,1] + 52.683;
   1:  PR[91,2] = PR[90,2] + -33.153;
   1:  PR[91,3] = PR[90,3] + 135.778;
   1:L PR[91] R[100]mm/sec CNT100;
   1:  PR[91,1] = PR[90,1] + 55.469;
   1:  PR[91,2] = PR[90,2] + -32.639;
   1:  PR[91,3] = PR[90,3] + 135.795;
   1:L PR[91] R[100]mm/sec CNT100;
   1:  PR[91,1] = PR[90,1] + 58.008;
   1:  PR[91,2] = PR[90,2] + -32.031;
   1:  PR[91,3] = PR[90,3] + 135.811;
   1:L PR[91] R[100]mm/sec CNT100;
   1:  PR[91,1] = PR[90,1] + 60.044;
   1:  PR[91,2] = PR[90,2] + -31.273;
   1:  PR[91,3] = PR[90,3] + 135.825;
   1:L PR[91] R[100]mm/sec CNT100;
   1:  PR[91,1] = PR[90,1] + 66.094;
   1:  PR[91,2] = PR[90,2] + -28.956;
   1:  PR[91,3] = PR[90,3] + 135.838;
   1:L PR[91] R[100]mm/sec CNT100;
   1:  PR[91,1] = PR[90,1] + 67.929;
   1:  PR[91,2] = PR[90,2] + -28.018;
   1:  PR[91,3] = PR[90,3] + 135.874;
   1:L PR[91] R[100]mm/sec CNT100;
   1:  PR[91,1] = PR[90,1] + 69.432;
   1:  PR[91,2] = PR[90,2] + -26.985;
   1:  PR[91,3] = PR[90,3] + 135.886;
   1:L PR[91] R[100]mm/sec CNT100;
   1:  PR[91,1] = PR[90,1] + 74.677;
   1:  PR[91,2] = PR[90,2] + -23.258;
   1:  PR[91,3] = PR[90,3] + 135.896;
   1:L PR[91] R[100]mm/sec CNT100;
   1:  PR[91,1] = PR[90,1] + 75.918;
   1:  PR[91,2] = PR[90,2] + -22.146;
   1:  PR[91,3] = PR[90,3] + 135.933;
   1:L PR[91] R[100]mm/sec CNT100;
   1:  PR[91,1] = PR[90,1] + 80.802;
   1:  PR[91,2] = PR[90,2] + -16.265;
   1:  PR[91,3] = PR[90,3] + 135.942;
   1:L PR[91] R[100]mm/sec CNT100;
   1:  PR[91,1] = PR[90,1] + 81.529;
   1:  PR[91,2] = PR[90,2] + -15.091;
   1:  PR[91,3] = PR[90,3] + 135.985;
   1:L PR[91] R[100]mm/sec CNT100;
   1:  PR[91,1] = PR[90,1] + 82.085;
   1:  PR[91,2] = PR[90,2] + -13.779;
   1:  PR[91,3] = PR[90,3] + 135.993;
   1:L PR[91] R[100]mm/sec CNT100;
   1:  PR[91,1] = PR[90,1] + 84.398;
   1:  PR[91,2] = PR[90,2] + -8.601;
   1:  PR[91,3] = PR[90,3] + 136.001;
   1:L PR[91] R[100]mm/sec CNT100;
   1:  PR[91,1] = PR[90,1] + 84.687;
   1:  PR[91,2] = PR[90,2] + -7.437;
   1:  PR[91,3] = PR[90,3] + 136.033;
   1:L PR[91] R[100]mm/sec CNT100;
   1:  PR[91,1] = PR[90,1] + 84.801;
   1:  PR[91,2] = PR[90,2] + -6.036;
   1:  PR[91,3] = PR[90,3] + 136.040;
   1:L PR[91] R[100]mm/sec CNT100;
   1:  PR[91,1] = PR[90,1] + 85.562;
   1:  PR[91,2] = PR[90,2] + -0.670;
   1:  PR[91,3] = PR[90,3] + 136.048;
